C03645=1237.341,-59.055,-37.494,-179.972,5.224,148.895
C03646=1237.346,-59.306,-37.482,-179.974,5.224,148.895
C03647=1237.351,-59.555,-37.469,-179.977,5.224,148.896
C03648=1237.356,-59.805,-37.457,-179.980,5.225,148.897
C03649=1237.361,-60.054,-37.445,-179.982,5.224,148.898
C03650=1237.367,-60.304,-37.433,-179.984,5.224,148.898
C03651=1237.371,-60.553,-37.421,-179.987,5.224,148.899
C03652=1237.376,-60.803,-37.408,-179.989,5.224,148.900
C03653=1237.382,-61.053,-37.396,-179.992,5.224,148.900
C03654=1237.387,-61.302,-37.384,-179.994,5.224,148.901
C03655=1237.392,-61.552,-37.371,-179.996,5.224,148.902
C03656=1237.397,-61.802,-37.359,-179.999,5.223,148.903
C03657=1237.402,-62.052,-37.347,179.999,5.224,148.903
C03658=1237.407,-62.301,-37.334,179.996,5.223,148.904
C03659=1237.412,-62.551,-37.323,179.994,5.223,148.905
C03660=1237.418,-62.801,-37.311,179.991,5.223,148.905
C03661=1237.423,-63.050,-37.299,179.989,5.223,148.906
C03662=1237.428,-63.300,-37.287,179.986,5.223,148.907
C03663=1237.433,-63.549,-37.274,179.984,5.223,148.908
C03664=1237.439,-63.799,-37.262,179.981,5.223,148.908
C03665=1237.443,-64.048,-37.250,179.979,5.223,148.909
C03666=1237.449,-64.298,-37.238,179.977,5.223,148.910
C03667=1237.454,-64.547,-37.226,179.974,5.223,148.911
C03668=1237.459,-64.797,-37.214,179.972,5.223,148.911
C03669=1237.464,-65.047,-37.202,179.970,5.223,148.912
C03670=1237.468,-65.297,-37.190,179.967,5.222,148.913
C03671=1237.474,-65.547,-37.178,179.965,5.223,148.913
C03672=1237.479,-65.796,-37.165,179.962,5.222,148.914
C03673=1237.484,-66.046,-37.153,179.960,5.223,148.915
C03674=1237.490,-66.296,-37.141,179.958,5.222,148.916
C03675=1237.494,-66.545,-37.129,179.955,5.223,148.916
C03676=1237.500,-66.795,-37.117,179.953,5.222,148.917
C03677=1237.505,-67.045,-37.106,179.951,5.222,148.918
C03678=1237.510,-67.294,-37.093,179.948,5.222,148.919
C03679=1237.515,-67.544,-37.082,179.945,5.223,148.919
C03680=1237.520,-67.794,-37.070,179.943,5.222,148.920
C03681=1237.525,-68.043,-37.057,179.941,5.222,148.921
C03682=1237.531,-68.293,-37.045,179.938,5.222,148.921
C03683=1237.535,-68.543,-37.034,179.936,5.222,148.922
C03684=1237.541,-68.792,-37.021,179.933,5.222,148.923
C03685=1237.546,-69.042,-37.010,179.931,5.221,148.924
C03686=1237.551,-69.292,-36.998,179.928,5.222,148.924
C03687=1237.556,-69.541,-36.986,179.926,5.221,148.925
C03688=1237.561,-69.791,-36.974,179.924,5.222,148.926
C03689=1237.567,-70.041,-36.962,179.921,5.221,148.926
C03690=1237.572,-70.291,-36.950,179.919,5.221,148.927
C03691=1237.576,-70.540,-36.938,179.916,5.221,148.928
C03692=1237.582,-70.789,-36.926,179.914,5.221,148.929
C03693=1237.588,-71.039,-36.915,179.912,5.221,148.929
C03694=1237.593,-71.289,-36.903,179.909,5.221,148.930
C03695=1237.598,-71.538,-36.891,179.906,5.221,148.931
C03696=1237.603,-71.788,-36.879,179.904,5.221,148.932
C03697=1237.608,-72.037,-36.867,179.902,5.221,148.932
C03698=1237.613,-72.287,-36.856,179.899,5.221,148.933
C03699=1237.619,-72.537,-36.844,179.897,5.221,148.934
C03700=1237.623,-72.786,-36.832,179.895,5.221,148.934
C03701=1237.629,-73.036,-36.820,179.892,5.221,148.935
C03702=1237.634,-73.286,-36.808,179.890,5.221,148.936
C03703=1237.639,-73.536,-36.797,179.887,5.220,148.937
C03704=1237.644,-73.786,-36.785,179.885,5.221,148.937
C03705=1237.650,-74.055,-36.772,179.882,5.220,148.938
C03706=1237.655,-74.326,-36.759,179.880,5.221,148.939
C03707=1237.661,-74.596,-36.746,179.877,5.221,148.940
C03708=1237.667,-74.866,-36.734,179.875,5.220,148.940
C03709=1237.672,-75.116,-36.722,179.872,5.220,148.941
C03710=1237.677,-75.365,-36.710,179.870,5.220,148.942
C03711=1237.682,-75.615,-36.699,179.868,5.220,148.942
C03712=1237.687,-75.865,-36.687,179.865,5.220,148.943
C03713=1237.692,-76.115,-36.675,179.863,5.220,148.944
C03714=1237.698,-76.365,-36.664,179.860,5.220,148.945
C03715=1237.702,-76.614,-36.652,179.858,5.220,148.945
C03716=1237.708,-76.864,-36.641,179.855,5.220,148.946
C03717=1237.713,-77.113,-36.629,179.853,5.220,148.947
C03718=1237.718,-77.363,-36.618,179.850,5.220,148.948
C03719=1237.723,-77.613,-36.606,179.848,5.220,148.948
C03720=1237.729,-77.863,-36.594,179.845,5.220,148.949
C03721=1237.733,-78.112,-36.583,179.843,5.220,148.950
C03722=1237.739,-78.362,-36.571,179.841,5.220,148.950
C03723=1237.744,-78.612,-36.559,179.839,5.220,148.951
C03724=1237.749,-78.861,-36.548,179.836,5.219,148.952
C03725=1237.755,-79.110,-36.536,179.834,5.220,148.953
C03726=1237.759,-79.360,-36.524,179.831,5.219,148.953
C03727=1237.765,-79.610,-36.513,179.829,5.220,148.954
C03728=1237.769,-79.860,-36.501,179.826,5.219,148.955
C03729=1237.775,-80.110,-36.489,179.824,5.220,148.955
C03730=1237.780,-80.359,-36.479,179.822,5.220,148.956
C03731=1237.786,-80.609,-36.467,179.820,5.219,148.957
C03732=1237.791,-80.859,-36.456,179.817,5.220,148.958
C03733=1237.796,-81.109,-36.444,179.815,5.219,148.958
C03734=1237.801,-81.358,-36.433,179.813,5.220,148.959
C03735=1237.806,-81.608,-36.421,179.810,5.219,148.960
C03736=1237.811,-81.857,-36.410,179.808,5.219,148.960
C03737=1237.816,-82.107,-36.399,179.805,5.219,148.961
C03738=1237.821,-82.357,-36.387,179.803,5.219,148.962
C03739=1237.826,-82.606,-36.376,179.800,5.219,148.963
C03740=1237.832,-82.856,-36.364,179.798,5.220,148.963
C03741=1237.837,-83.105,-36.353,179.795,5.219,148.964
C03742=1237.842,-83.355,-36.341,179.793,5.220,148.965
C03743=1237.847,-83.605,-36.330,179.790,5.219,148.966
C03744=1237.853,-83.855,-36.318,179.788,5.219,148.966
C03745=1237.857,-84.105,-36.307,179.786,5.219,148.967
C03746=1237.863,-84.354,-36.296,179.784,5.219,148.968
C03747=1237.868,-84.604,-36.284,179.781,5.219,148.968
C03748=1237.873,-84.853,-36.273,179.779,5.219,148.969
C03749=1237.878,-85.103,-36.261,179.776,5.219,148.970
C03750=1237.883,-85.353,-36.250,179.774,5.219,148.971
C03751=1237.889,-85.603,-36.240,179.771,5.219,148.971
C03752=1237.894,-85.852,-36.228,179.769,5.219,148.972
C03753=1237.899,-86.102,-36.216,179.767,5.218,148.973
C03754=1237.903,-86.352,-36.205,179.765,5.219,148.973
C03755=1237.909,-86.601,-36.194,179.762,5.218,148.974
C03756=1237.914,-86.851,-36.182,179.760,5.219,148.975
C03757=1237.920,-87.101,-36.171,179.757,5.218,148.976
C03758=1237.925,-87.351,-36.160,179.755,5.219,148.976
C03759=1237.930,-87.600,-36.149,179.752,5.218,148.977
C03760=1237.935,-87.850,-36.137,179.750,5.218,148.978
C03761=1237.940,-88.100,-36.127,179.748,5.219,148.978
C03762=1237.945,-88.349,-36.115,179.745,5.218,148.979
C03763=1237.951,-88.599,-36.104,179.743,5.219,148.980
C03764=1237.956,-88.848,-36.092,179.741,5.218,148.981
C03765=1237.961,-89.099,-36.082,179.739,5.219,148.981
C03766=1237.966,-89.349,-36.070,179.736,5.218,148.982
C03767=1237.971,-89.597,-36.059,179.734,5.218,148.983
C03768=1237.976,-89.847,-36.048,179.731,5.218,148.983
C03769=1237.982,-90.098,-36.037,179.729,5.218,148.984
C03770=1237.987,-90.347,-36.026,179.726,5.218,148.985
C03771=1237.992,-90.596,-36.014,179.724,5.218,148.985
C03772=1237.997,-90.846,-36.004,179.722,5.218,148.986
C03773=1238.003,-91.096,-35.992,179.720,5.218,148.987
C03774=1238.008,-91.345,-35.981,179.716,5.218,148.988
C03775=1238.013,-91.596,-35.970,179.714,5.218,148.989
C03776=1238.018,-91.845,-35.959,179.712,5.218,148.989
C03777=1238.023,-92.094,-35.948,179.710,5.218,148.990
C03778=1238.028,-92.345,-35.937,179.707,5.218,148.991
C03779=1238.033,-92.594,-35.926,179.705,5.218,148.991
C03780=1238.039,-92.843,-35.914,179.702,5.218,148.992
C03781=1238.044,-93.094,-35.904,179.700,5.218,148.993
C03782=1238.049,-93.343,-35.892,179.698,5.218,148.994
C03783=1238.054,-93.593,-35.882,179.695,5.218,148.994
C03784=1238.060,-93.843,-35.870,179.693,5.218,148.995
C03785=1238.064,-94.092,-35.859,179.690,5.218,148.996
C03786=1238.070,-94.342,-35.849,179.688,5.218,148.996
C03787=1238.075,-94.592,-35.837,179.686,5.218,148.997
C03788=1238.080,-94.841,-35.827,179.684,5.218,148.998
C03789=1238.086,-95.091,-35.815,179.681,5.218,148.999
C03790=1238.090,-95.341,-35.804,179.679,5.218,148.999
C03791=1238.096,-95.590,-35.794,179.676,5.218,149.000
C03792=1238.101,-95.840,-35.783,179.674,5.218,149.001
C03793=1238.106,-96.090,-35.772,179.671,5.217,149.001
C03794=1238.112,-96.339,-35.760,179.669,5.218,149.002
C03795=1238.117,-96.590,-35.750,179.667,5.217,149.003
C03796=1238.122,-96.839,-35.739,179.665,5.218,149.004
C03797=1238.127,-97.089,-35.728,179.662,5.218,149.004
C03798=1238.132,-97.338,-35.717,179.660,5.218,149.005
C03799=1238.137,-97.588,-35.707,179.658,5.218,149.006
C03800=1238.143,-97.838,-35.695,179.655,5.217,149.006
C03801=1238.148,-98.088,-35.684,179.653,5.218,149.007
C03802=1238.153,-98.337,-35.674,179.650,5.217,149.008
C03803=1238.158,-98.587,-35.663,179.648,5.218,149.009
C03804=1238.163,-98.836,-35.652,179.645,5.217,149.009
C03805=1238.168,-99.087,-35.641,179.643,5.218,149.010
C03806=1238.174,-99.335,-35.631,179.641,5.217,149.011
C03807=1238.179,-99.586,-35.619,179.639,5.218,149.011
C03808=1238.184,-99.836,-35.608,179.636,5.217,149.012
C03809=1238.190,-100.106,-35.598,179.634,5.217,149.013
C03810=1238.195,-100.377,-35.585,179.631,5.217,149.014
C03811=1238.200,-100.648,-35.574,179.629,5.218,149.014
C03812=1238.207,-100.919,-35.562,179.626,5.217,149.015
C03813=1238.212,-101.168,-35.551,179.624,5.218,149.016
C03814=1238.217,-101.419,-35.541,179.621,5.217,149.017
C03815=1238.222,-101.668,-35.530,179.619,5.218,149.017
C03816=1238.227,-101.918,-35.519,179.616,5.217,149.018
C03817=1238.232,-102.167,-35.509,179.614,5.217,149.019
C03818=1238.238,-102.417,-35.497,179.612,5.217,149.019
C03819=1238.243,-102.667,-35.487,179.609,5.217,149.020
C03820=1238.248,-102.917,-35.476,179.607,5.217,149.021
C03821=1238.254,-103.166,-35.465,179.605,5.217,149.022
C03822=1238.259,-103.416,-35.455,179.602,5.217,149.022
C03823=1238.264,-103.666,-35.444,179.600,5.217,149.023
C03824=1238.269,-103.915,-35.433,179.598,5.218,149.024
C03825=1238.275,-104.165,-35.423,179.595,5.217,149.024
C03826=1238.280,-104.415,-35.412,179.593,5.217,149.025
C03827=1238.284,-104.665,-35.401,179.590,5.217,149.026
C03828=1238.290,-104.914,-35.391,179.588,5.217,149.027
C03829=1238.295,-105.165,-35.380,179.586,5.217,149.027
C03830=1238.300,-105.414,-35.369,179.584,5.217,149.028
C03831=1238.305,-105.664,-35.359,179.581,5.217,149.029
C03832=1238.311,-105.913,-35.349,179.579,5.217,149.029
C03833=1238.316,-106.164,-35.338,179.576,5.217,149.030
C03834=1238.321,-106.412,-35.327,179.574,5.217,149.031
C03835=1238.326,-106.663,-35.317,179.572,5.217,149.031
C03836=1238.332,-106.912,-35.306,179.570,5.217,149.032
C03837=1238.337,-107.163,-35.296,179.568,5.217,149.033
C03838=1238.342,-107.411,-35.285,179.565,5.217,149.034
C03839=1238.348,-107.661,-35.275,179.563,5.217,149.034
C03840=1238.353,-107.911,-35.264,179.560,5.216,149.035
C03841=1238.358,-108.161,-35.254,179.558,5.217,149.036
C03842=1238.362,-108.410,-35.243,179.555,5.216,149.036
C03843=1238.368,-108.660,-35.233,179.553,5.217,149.037
C03844=1238.373,-108.910,-35.222,179.551,5.216,149.038
C03845=1238.378,-109.159,-35.212,179.549,5.217,149.039
C03846=1238.383,-109.410,-35.202,179.546,5.217,149.039
C03847=1238.389,-109.659,-35.191,179.544,5.217,149.040
C03848=1238.394,-109.909,-35.180,179.542,5.217,149.041
C03849=1238.399,-110.158,-35.170,179.539,5.217,149.041
C03850=1238.404,-110.409,-35.159,179.537,5.217,149.042
C03851=1238.410,-110.658,-35.149,179.534,5.216,149.043
C03852=1238.415,-110.908,-35.139,179.532,5.217,149.044
C03853=1238.420,-111.158,-35.128,179.529,5.216,149.044
C03854=1238.425,-111.407,-35.119,179.527,5.217,149.045
C03855=1238.430,-111.657,-35.107,179.525,5.217,149.046
C03856=1238.436,-111.906,-35.097,179.523,5.217,149.046
C03857=1238.441,-112.157,-35.087,179.520,5.217,149.047
C03858=1238.446,-112.406,-35.076,179.518,5.217,149.048
C03859=1238.452,-112.656,-35.066,179.516,5.217,149.049
C03860=1238.457,-112.906,-35.056,179.513,5.216,149.049
C03861=1238.462,-113.155,-35.045,179.511,5.217,149.050
C03862=1238.467,-113.405,-35.035,179.508,5.216,149.051
C03863=1238.472,-113.655,-35.025,179.506,5.217,149.051
C03864=1238.478,-113.904,-35.015,179.503,5.216,149.052
C03865=1238.483,-114.155,-35.004,179.501,5.217,149.053
C03866=1238.488,-114.404,-34.994,179.500,5.217,149.053
C03867=1238.494,-114.653,-34.983,179.497,5.216,149.054
C03868=1238.498,-114.903,-34.973,179.495,5.217,149.055
C03869=1238.504,-115.153,-34.963,179.492,5.216,149.055
C03870=1238.509,-115.403,-34.953,179.490,5.217,149.056
C03871=1238.514,-115.652,-34.942,179.488,5.216,149.057
C03872=1238.520,-115.902,-34.932,179.485,5.216,149.058
C03873=1238.524,-116.152,-34.922,179.483,5.216,149.058
C03874=1238.530,-116.401,-34.912,179.481,5.216,149.059
C03875=1238.535,-116.651,-34.902,179.479,5.217,149.060
C03876=1238.540,-116.901,-34.891,179.476,5.216,149.060
C03877=1238.546,-117.151,-34.881,179.474,5.217,149.061
C03878=1238.550,-117.401,-34.871,179.471,5.216,149.062
C03879=1238.556,-117.651,-34.861,179.469,5.217,149.063
C03880=1238.562,-117.900,-34.851,179.466,5.216,149.063
C03881=1238.567,-118.151,-34.841,179.464,5.217,149.064
C03882=1238.571,-118.400,-34.831,179.462,5.216,149.065
C03883=1238.577,-118.649,-34.821,179.459,5.216,149.065
C03884=1238.582,-118.900,-34.810,179.457,5.217,149.066
C03885=1238.588,-119.149,-34.800,179.455,5.216,149.067
C03886=1238.592,-119.398,-34.790,179.453,5.216,149.067
C03887=1238.597,-119.649,-34.780,179.450,5.216,149.068
C03888=1238.603,-119.898,-34.770,179.448,5.216,149.069
C03889=1238.608,-120.148,-34.760,179.446,5.216,149.070
C03890=1238.613,-120.397,-34.750,179.444,5.216,149.070
C03891=1238.619,-120.648,-34.740,179.441,5.216,149.071
C03892=1238.624,-120.897,-34.730,179.439,5.216,149.072
C03893=1238.629,-121.147,-34.720,179.437,5.217,149.072
C03894=1238.634,-121.397,-34.710,179.434,5.216,149.073
C03895=1238.640,-121.646,-34.699,179.432,5.216,149.074
C03896=1238.645,-121.896,-34.690,179.429,5.216,149.075
C03897=1238.650,-122.146,-34.679,179.427,5.216,149.075
C03898=1238.656,-122.396,-34.670,179.424,5.216,149.076
C03899=1238.660,-122.645,-34.660,179.422,5.216,149.077
C03900=1238.666,-122.895,-34.650,179.421,5.216,149.077
C03901=1238.671,-123.145,-34.639,179.418,5.216,149.078
C03902=1238.676,-123.394,-34.630,179.416,5.216,149.079
C03903=1238.682,-123.644,-34.620,179.413,5.216,149.079
C03904=1238.687,-123.895,-34.610,179.411,5.216,149.080
C03905=1238.692,-124.144,-34.600,179.408,5.216,149.081
C03906=1238.697,-124.394,-34.590,179.406,5.216,149.082
C03907=1238.702,-124.643,-34.580,179.404,5.216,149.082
C03908=1238.707,-124.894,-34.570,179.402,5.216,149.083
C03909=1238.713,-125.143,-34.560,179.400,5.216,149.084
C03910=1238.718,-125.392,-34.551,179.397,5.216,149.084
C03911=1238.724,-125.642,-34.540,179.395,5.216,149.085
C03912=1238.729,-125.893,-34.530,179.393,5.216,149.086
C03913=1238.307,-125.903,-34.566,179.388,5.219,149.088
C03914=1238.302,-125.653,-34.575,179.391,5.220,149.087
C03915=1238.297,-125.403,-34.586,179.393,5.219,149.086
C03916=1238.292,-125.154,-34.595,179.395,5.219,149.086
C03917=1238.286,-124.904,-34.605,179.397,5.220,149.085
C03918=1238.280,-124.654,-34.615,179.399,5.219,149.084
C03919=1238.276,-124.404,-34.625,179.402,5.220,149.084
C03920=1238.270,-124.154,-34.635,179.404,5.219,149.083
C03921=1238.265,-123.905,-34.645,179.407,5.220,149.082
C03922=1238.260,-123.655,-34.654,179.409,5.219,149.081
C03923=1238.255,-123.405,-34.665,179.411,5.220,149.081
C03924=1238.250,-123.156,-34.674,179.414,5.219,149.080
C03925=1238.244,-122.906,-34.685,179.416,5.219,149.079
C03926=1238.239,-122.656,-34.695,179.418,5.219,149.079
C03927=1238.234,-122.406,-34.704,179.420,5.219,149.078
C03928=1238.228,-122.156,-34.714,179.423,5.220,149.077
C03929=1238.223,-121.907,-34.724,179.425,5.220,149.077
C03930=1238.219,-121.657,-34.734,179.427,5.220,149.076
C03931=1238.213,-121.407,-34.745,179.429,5.220,149.075
C03932=1238.207,-121.158,-34.755,179.432,5.220,149.075
C03933=1238.201,-120.908,-34.764,179.434,5.220,149.074
C03934=1238.197,-120.658,-34.774,179.436,5.219,149.073
C03935=1238.192,-120.408,-34.785,179.439,5.220,149.072
C03936=1238.186,-120.159,-34.795,179.441,5.219,149.072
C03937=1238.182,-119.909,-34.805,179.444,5.220,149.071
C03938=1238.176,-119.659,-34.815,179.446,5.219,149.070
C03939=1238.171,-119.410,-34.825,179.449,5.220,149.070
C03940=1238.166,-119.159,-34.836,179.451,5.220,149.069
C03941=1238.161,-118.910,-34.845,179.453,5.219,149.068
C03942=1238.155,-118.660,-34.855,179.455,5.220,149.067
C03943=1238.150,-118.410,-34.865,179.458,5.219,149.067
C03944=1238.145,-118.161,-34.875,179.460,5.220,149.066
C03945=1238.139,-117.911,-34.885,179.462,5.220,149.065
C03946=1238.134,-117.661,-34.896,179.465,5.220,149.065
C03947=1238.129,-117.411,-34.906,179.467,5.220,149.064
C03948=1238.124,-117.162,-34.916,179.469,5.220,149.063
C03949=1238.119,-116.912,-34.926,179.471,5.220,149.063
C03950=1238.113,-116.662,-34.936,179.473,5.219,149.062
C03951=1238.108,-116.413,-34.947,179.476,5.220,149.061
C03952=1238.103,-116.162,-34.957,179.478,5.220,149.060
C03953=1238.098,-115.913,-34.967,179.481,5.220,149.060
C03954=1238.092,-115.664,-34.977,179.483,5.220,149.059
C03955=1238.087,-115.413,-34.988,179.486,5.220,149.058
C03956=1238.082,-115.164,-34.998,179.488,5.220,149.058
C03957=1238.077,-114.914,-35.008,179.491,5.220,149.057
C03958=1238.072,-114.664,-35.018,179.493,5.220,149.056
C03959=1238.066,-114.415,-35.028,179.495,5.220,149.055
C03960=1238.061,-114.165,-35.039,179.497,5.220,149.055
C03961=1238.056,-113.915,-35.049,179.499,5.219,149.054
C03962=1238.050,-113.665,-35.059,179.502,5.220,149.053
C03963=1238.045,-113.415,-35.070,179.504,5.220,149.053
C03964=1238.040,-113.166,-35.079,179.506,5.220,149.052
C03965=1238.035,-112.916,-35.090,179.509,5.220,149.051
C03966=1238.030,-112.667,-35.101,179.511,5.220,149.051
C03967=1238.024,-112.417,-35.111,179.513,5.220,149.050
C03968=1238.019,-112.167,-35.122,179.516,5.220,149.049
C03969=1238.014,-111.917,-35.132,179.518,5.220,149.049
C03970=1238.009,-111.667,-35.142,179.520,5.220,149.048
C03971=1238.004,-111.418,-35.152,179.523,5.220,149.047
C03972=1237.999,-111.168,-35.163,179.525,5.220,149.046
C03973=1237.993,-110.918,-35.173,179.528,5.220,149.046
C03974=1237.988,-110.669,-35.183,179.530,5.220,149.045
C03975=1237.983,-110.419,-35.194,179.532,5.220,149.044
C03976=1237.977,-110.170,-35.205,179.534,5.220,149.044
C03977=1237.972,-109.919,-35.215,179.537,5.220,149.043
C03978=1237.967,-109.670,-35.225,179.539,5.220,149.042
C03979=1237.962,-109.419,-35.236,179.541,5.220,149.041
C03980=1237.956,-109.170,-35.246,179.544,5.220,149.041
C03981=1237.952,-108.921,-35.256,179.546,5.220,149.040
C03982=1237.947,-108.671,-35.267,179.549,5.220,149.039
C03983=1237.941,-108.422,-35.277,179.551,5.220,149.038
C03984=1237.936,-108.171,-35.288,179.554,5.220,149.038
C03985=1237.930,-107.922,-35.298,179.556,5.220,149.037
C03986=1237.926,-107.672,-35.309,179.558,5.220,149.036
C03987=1237.920,-107.423,-35.320,179.560,5.220,149.036
C03988=1237.915,-107.172,-35.330,179.563,5.220,149.035
C03989=1237.909,-106.923,-35.340,179.565,5.220,149.034
C03990=1237.904,-106.673,-35.351,179.567,5.220,149.033
C03991=1237.899,-106.424,-35.362,179.570,5.220,149.033
C03992=1237.894,-106.173,-35.372,179.572,5.220,149.032
C03993=1237.889,-105.924,-35.383,179.574,5.221,149.032
C03994=1237.884,-105.674,-35.394,179.576,5.220,149.031
C03995=1237.878,-105.425,-35.404,179.579,5.221,149.030
C03996=1237.873,-105.174,-35.415,179.581,5.220,149.029
C03997=1237.868,-104.925,-35.425,179.584,5.221,149.029
C03998=1237.863,-104.675,-35.436,179.586,5.221,149.028
C03999=1237.857,-104.426,-35.446,179.589,5.221,149.027
C04000=1237.852,-104.175,-35.457,179.591,5.221,149.027
C04001=1237.847,-103.927,-35.468,179.593,5.221,149.026
C04002=1237.842,-103.676,-35.478,179.595,5.221,149.025
C04003=1237.836,-103.427,-35.489,179.598,5.220,149.024
C04004=1237.832,-103.177,-35.500,179.600,5.221,149.024
C04005=1237.826,-102.928,-35.510,179.602,5.220,149.023
C04006=1237.821,-102.677,-35.521,179.605,5.221,149.022
C04007=1237.816,-102.428,-35.532,179.607,5.221,149.022
C04008=1237.811,-102.178,-35.542,179.610,5.221,149.021
C04009=1237.806,-101.928,-35.553,179.612,5.221,149.020
C04010=1237.801,-101.679,-35.564,179.615,5.221,149.019
C04011=1237.796,-101.429,-35.574,179.617,5.221,149.019
C04012=1237.790,-101.180,-35.585,179.619,5.221,149.018
C04013=1237.785,-100.929,-35.596,179.621,5.221,149.017
C04014=1237.779,-100.659,-35.608,179.624,5.221,149.017
C04015=1237.773,-100.388,-35.619,179.627,5.220,149.016
C04016=1237.768,-100.117,-35.631,179.629,5.221,149.015
C04017=1237.763,-99.846,-35.643,179.631,5.221,149.014
C04018=1237.757,-99.597,-35.653,179.634,5.221,149.013
C04019=1237.752,-99.347,-35.665,179.636,5.221,149.013
C04020=1237.747,-99.097,-35.675,179.639,5.221,149.012
C04021=1237.742,-98.847,-35.685,179.641,5.221,149.011
C04022=1237.736,-98.598,-35.697,179.644,5.221,149.011
C04023=1237.731,-98.348,-35.708,179.646,5.221,149.010
C04024=1237.726,-98.098,-35.719,179.648,5.221,149.009
C04025=1237.720,-97.848,-35.729,179.651,5.221,149.009
C04026=1237.716,-97.599,-35.740,179.653,5.221,149.008
C04027=1237.710,-97.349,-35.751,179.655,5.221,149.007
C04028=1237.706,-97.100,-35.762,179.657,5.221,149.006
C04029=1237.700,-96.849,-35.773,179.660,5.221,149.006
C04030=1237.694,-96.600,-35.784,179.662,5.221,149.005
C04031=1237.689,-96.350,-35.794,179.665,5.221,149.004
C04032=1237.685,-96.100,-35.806,179.667,5.221,149.004
C04033=1237.679,-95.851,-35.816,179.670,5.221,149.003
C04034=1237.674,-95.601,-35.828,179.672,5.221,149.002
C04035=1237.668,-95.352,-35.839,179.674,5.221,149.001
C04036=1237.663,-95.102,-35.849,179.676,5.221,149.001
C04037=1237.659,-94.852,-35.861,179.679,5.222,149.000
C04038=1237.653,-94.602,-35.871,179.681,5.221,148.999
C04039=1237.648,-94.353,-35.883,179.684,5.222,148.999
C04040=1237.643,-94.102,-35.893,179.686,5.221,148.998
C04041=1237.637,-93.853,-35.904,179.689,5.222,148.997
C04042=1237.633,-93.604,-35.916,179.691,5.221,148.996
C04043=1237.628,-93.353,-35.926,179.693,5.222,148.996
C04044=1237.622,-93.104,-35.938,179.696,5.222,148.995
C04045=1237.617,-92.854,-35.948,179.698,5.221,148.994
C04046=1237.612,-92.604,-35.959,179.700,5.222,148.994
C04047=1237.607,-92.355,-35.970,179.702,5.221,148.993
C04048=1237.601,-92.105,-35.982,179.705,5.222,148.992
C04049=1237.596,-91.855,-35.993,179.707,5.221,148.991
C04050=1237.591,-91.606,-36.004,179.710,5.222,148.991
C04051=1237.585,-91.356,-36.015,179.712,5.222,148.990
C04052=1237.581,-91.106,-36.026,179.715,5.222,148.989
C04053=1237.575,-90.857,-36.037,179.717,5.222,148.989
C04054=1237.570,-90.607,-36.048,179.719,5.222,148.988
C04055=1237.565,-90.357,-36.060,179.721,5.222,148.987
C04056=1237.560,-90.108,-36.071,179.724,5.222,148.986
C04057=1237.555,-89.858,-36.081,179.726,5.222,148.986
C04058=1237.549,-89.608,-36.093,179.729,5.222,148.985
C04059=1237.544,-89.358,-36.104,179.731,5.222,148.984
C04060=1237.539,-89.109,-36.115,179.734,5.222,148.984
C04061=1237.534,-88.859,-36.126,179.736,5.222,148.983
C04062=1237.529,-88.609,-36.138,179.739,5.222,148.982
C04063=1237.523,-88.360,-36.149,179.741,5.222,148.981
C04064=1237.518,-88.110,-36.159,179.743,5.221,148.981
C04065=1237.513,-87.860,-36.171,179.746,5.222,148.980
C04066=1237.508,-87.611,-36.182,179.748,5.222,148.979
C04067=1237.502,-87.361,-36.194,179.751,5.222,148.978
C04068=1237.498,-87.112,-36.205,179.753,5.222,148.978
C04069=1237.493,-86.861,-36.216,179.755,5.222,148.977
C04070=1237.487,-86.611,-36.228,179.757,5.222,148.976
C04071=1237.482,-86.363,-36.239,179.760,5.222,148.976
C04072=1237.477,-86.113,-36.250,179.762,5.222,148.975
C04073=1237.472,-85.863,-36.262,179.765,5.222,148.974
C04074=1237.467,-85.613,-36.272,179.767,5.222,148.973
C04075=1237.461,-85.364,-36.283,179.770,5.222,148.973
C04076=1237.456,-85.114,-36.295,179.772,5.222,148.972
C04077=1237.451,-84.864,-36.306,179.774,5.223,148.971
C04078=1237.446,-84.614,-36.318,179.776,5.222,148.971
C04079=1237.441,-84.365,-36.330,179.779,5.223,148.970
C04080=1237.436,-84.115,-36.340,179.781,5.222,148.969
C04081=1237.430,-83.865,-36.352,179.784,5.223,148.968
C04082=1237.426,-83.616,-36.363,179.786,5.222,148.968
C04083=1237.420,-83.366,-36.375,179.789,5.223,148.967
C04084=1237.415,-83.117,-36.386,179.791,5.223,148.966
C04085=1237.409,-82.867,-36.398,179.793,5.223,148.966
C04086=1237.405,-82.617,-36.409,179.796,5.223,148.965
C04087=1237.400,-82.368,-36.420,179.798,5.223,148.964
C04088=1237.395,-82.118,-36.432,179.800,5.223,148.963
C04089=1237.390,-81.867,-36.443,179.803,5.223,148.963
C04090=1237.384,-81.618,-36.454,179.805,5.223,148.962
C04091=1237.379,-81.368,-36.466,179.808,5.223,148.961
C04092=1237.373,-81.119,-36.477,179.810,5.223,148.961
C04093=1237.369,-80.869,-36.489,179.812,5.224,148.960
C04094=1237.363,-80.619,-36.501,179.815,5.223,148.959
C04095=1237.358,-80.370,-36.511,179.818,5.223,148.958
C04096=1237.353,-80.120,-36.523,179.820,5.223,148.958
C04097=1237.348,-79.871,-36.535,179.823,5.223,148.957
C04098=1237.342,-79.621,-36.547,179.825,5.223,148.956
C04099=1237.338,-79.371,-36.558,179.827,5.223,148.955
C04100=1237.332,-79.121,-36.570,179.829,5.223,148.955
C04101=1237.328,-78.871,-36.581,179.831,5.223,148.954
C04102=1237.322,-78.622,-36.593,179.834,5.223,148.953
C04103=1237.317,-78.373,-36.604,179.836,5.223,148.953
C04104=1237.311,-78.123,-36.616,179.839,5.223,148.952
C04105=1237.307,-77.873,-36.627,179.841,5.223,148.951
C04106=1237.301,-77.623,-36.639,179.844,5.224,148.950
C04107=1237.297,-77.373,-36.650,179.846,5.223,148.950
C04108=1237.291,-77.123,-36.662,179.848,5.224,148.949
C04109=1237.285,-76.874,-36.674,179.851,5.223,148.948
C04110=1237.281,-76.625,-36.685,179.853,5.224,148.948
C04111=1237.275,-76.375,-36.697,179.855,5.224,148.947
C04112=1237.271,-76.126,-36.709,179.858,5.224,148.946
C04113=1237.265,-75.876,-36.721,179.860,5.224,148.945
C04114=1237.261,-75.626,-36.732,179.863,5.224,148.945
C04115=1237.255,-75.376,-36.744,179.865,5.224,148.944
C04116=1237.250,-75.126,-36.756,179.867,5.224,148.943
C04117=1237.245,-74.877,-36.767,179.870,5.224,148.943
C04118=1237.239,-74.607,-36.780,179.873,5.224,148.942
C04119=1237.234,-74.337,-36.793,179.875,5.224,148.941
C04120=1237.228,-74.066,-36.804,179.877,5.224,148.940
C04121=1237.222,-73.796,-36.817,179.881,5.224,148.939
C04122=1237.217,-73.546,-36.829,179.883,5.224,148.939
C04123=1237.212,-73.297,-36.842,179.885,5.224,148.938
C04124=1237.207,-73.047,-36.853,179.888,5.224,148.937
C04125=1237.202,-72.797,-36.865,179.890,5.225,148.937
C04126=1237.197,-72.548,-36.876,179.892,5.224,148.936
C04127=1237.191,-72.298,-36.888,179.895,5.225,148.935
C04128=1237.186,-72.048,-36.900,179.897,5.224,148.934
C04129=1237.182,-71.799,-36.912,179.900,5.225,148.934
C04130=1237.176,-71.549,-36.924,179.902,5.224,148.933
C04131=1237.170,-71.299,-36.936,179.904,5.225,148.932
C04132=1237.165,-71.050,-36.947,179.907,5.225,148.932
C04133=1237.160,-70.801,-36.959,179.909,5.225,148.931
C04134=1237.155,-70.551,-36.971,179.911,5.225,148.930
C04135=1237.150,-70.301,-36.983,179.914,5.225,148.929
C04136=1237.145,-70.051,-36.994,179.917,5.226,148.929
C04137=1237.140,-69.802,-37.007,179.919,5.225,148.928
C04138=1237.134,-69.552,-37.019,179.922,5.225,148.927
C04139=1237.130,-69.302,-37.030,179.924,5.225,148.926
C04140=1237.124,-69.052,-37.042,179.927,5.226,148.926
C04141=1237.119,-68.803,-37.055,179.929,5.225,148.925
C04142=1237.114,-68.553,-37.067,179.931,5.226,148.924
C04143=1237.109,-68.303,-37.078,179.934,5.225,148.924
C04144=1237.104,-68.054,-37.091,179.936,5.226,148.923
C04145=1237.098,-67.804,-37.102,179.938,5.226,148.922
C04146=1237.093,-67.554,-37.114,179.941,5.226,148.921
C04147=1237.088,-67.305,-37.126,179.943,5.226,148.921
C04148=1237.083,-67.055,-37.138,179.946,5.226,148.920
C04149=1237.078,-66.805,-37.150,179.948,5.226,148.919
C04150=1237.073,-66.556,-37.163,179.950,5.226,148.919
C04151=1237.068,-66.306,-37.174,179.953,5.226,148.918
C04152=1237.062,-66.056,-37.186,179.955,5.226,148.917
C04153=1237.057,-65.807,-37.198,179.957,5.226,148.916
C04154=1237.052,-65.557,-37.210,179.960,5.227,148.916
C04155=1237.046,-65.307,-37.222,179.963,5.226,148.915
C04156=1237.042,-65.058,-37.234,179.965,5.226,148.914
C04157=1237.037,-64.808,-37.246,179.967,5.226,148.913
C04158=1237.032,-64.559,-37.259,179.970,5.227,148.913
C04159=1237.026,-64.309,-37.271,179.972,5.226,148.912
C04160=1237.021,-64.059,-37.282,179.975,5.227,148.911
C04161=1237.016,-63.810,-37.294,179.977,5.226,148.911
C04162=1237.011,-63.559,-37.307,179.980,5.227,148.910
C04163=1237.006,-63.310,-37.319,179.982,5.227,148.909
C04164=1237.001,-63.060,-37.331,179.984,5.227,148.908
C04165=1236.996,-62.811,-37.344,179.986,5.227,148.908
C04166=1236.990,-62.561,-37.356,179.989,5.227,148.907
C04167=1236.986,-62.312,-37.368,179.992,5.228,148.906
C04168=1236.981,-62.062,-37.380,179.994,5.227,148.906
C04169=1236.975,-61.813,-37.392,179.996,5.228,148.905
C04170=1236.970,-61.563,-37.404,179.999,5.227,148.904
C04171=1236.965,-61.313,-37.416,-179.998,5.228,148.903
C04172=1236.959,-61.063,-37.429,-179.996,5.227,148.903
C04173=1236.954,-60.814,-37.441,-179.994,5.228,148.902
C04174=1236.949,-60.563,-37.453,-179.991,5.227,148.901
C04175=1236.945,-60.314,-37.465,-179.989,5.228,148.900
C04176=1236.940,-60.065,-37.477,-179.987,5.228,148.900
C04177=1236.935,-59.815,-37.490,-179.984,5.228,148.899
C04178=1236.929,-59.565,-37.502,-179.982,5.228,148.898
C04179=1236.924,-59.316,-37.514,-179.979,5.228,148.898
C04180=1236.919,-59.066,-37.526,-179.977,5.228,148.897
C04181=1236.913,-58.817,-37.539,-179.975,5.228,148.896
C04182=1236.908,-58.567,-37.551,-179.972,5.228,148.896
C04183=1236.903,-58.317,-37.564,-179.970,5.228,148.895
C04184=1236.898,-58.067,-37.576,-179.967,5.229,148.894
C04185=1236.893,-57.818,-37.588,-179.965,5.229,148.893
C04186=1236.888,-57.568,-37.601,-179.962,5.229,148.893
C04187=1236.883,-57.319,-37.612,-179.960,5.228,148.892
C04188=1236.878,-57.069,-37.625,-179.957,5.229,148.891
C04189=1236.873,-56.820,-37.637,-179.955,5.229,148.890
C04190=1236.868,-56.569,-37.650,-179.952,5.229,148.890
C04191=1236.863,-56.320,-37.662,-179.950,5.229,148.889
C04192=1236.858,-56.071,-37.675,-179.948,5.229,148.888
C04193=1236.852,-55.821,-37.687,-179.945,5.229,148.888
C04194=1236.847,-55.571,-37.699,-179.943,5.229,148.887
C04195=1236.842,-55.322,-37.712,-179.941,5.229,148.886
C04196=1236.837,-55.071,-37.724,-179.938,5.230,148.885
C04197=1236.832,-54.822,-37.737,-179.936,5.229,148.885
C04198=1236.827,-54.573,-37.749,-179.933,5.230,148.884
C04199=1236.822,-54.323,-37.761,-179.931,5.230,148.883
C04200=1236.816,-54.074,-37.774,-179.929,5.230,148.883
C04201=1236.812,-53.824,-37.787,-179.925,5.230,148.882
C04202=1236.807,-53.574,-37.799,-179.923,5.230,148.881
C04203=1236.801,-53.324,-37.811,-179.921,5.230,148.880
C04204=1236.796,-53.075,-37.824,-179.919,5.230,148.880
C04205=1236.791,-52.826,-37.836,-179.916,5.230,148.879
C04206=1236.787,-52.576,-37.849,-179.914,5.230,148.878
C04207=1236.781,-52.326,-37.861,-179.911,5.231,148.877
C04208=1236.775,-52.076,-37.875,-179.909,5.230,148.877
C04209=1236.770,-51.827,-37.887,-179.906,5.231,148.876
C04210=1236.765,-51.577,-37.900,-179.904,5.231,148.875
C04211=1236.760,-51.327,-37.912,-179.902,5.231,148.875
C04212=1236.755,-51.077,-37.925,-179.899,5.231,148.874
C04213=1236.750,-50.828,-37.937,-179.897,5.231,148.873
C04214=1236.745,-50.579,-37.950,-179.894,5.232,148.873
C04215=1236.740,-50.329,-37.963,-179.892,5.231,148.872
C04216=1236.735,-50.079,-37.975,-179.889,5.231,148.871
C04217=1236.730,-49.830,-37.987,-179.887,5.231,148.870
C04218=1236.725,-49.580,-38.000,-179.884,5.231,148.870
C04219=1236.719,-49.330,-38.013,-179.882,5.231,148.869
C04220=1236.714,-49.081,-38.026,-179.879,5.232,148.868
C04221=1236.709,-48.831,-38.039,-179.877,5.232,148.867
C04222=1236.704,-48.561,-38.052,-179.875,5.232,148.867
C04223=1236.698,-48.292,-38.065,-179.872,5.232,148.866
C04224=1236.693,-48.022,-38.079,-179.869,5.232,148.865
C04225=1236.688,-47.752,-38.093,-179.867,5.232,148.864
C04226=1236.682,-47.503,-38.106,-179.864,5.233,148.864
C04227=1236.677,-47.253,-38.119,-179.862,5.232,148.863
C04228=1236.672,-47.003,-38.132,-179.859,5.233,148.862
C04229=1236.667,-46.754,-38.144,-179.856,5.233,148.861
C04230=1236.662,-46.505,-38.157,-179.854,5.233,148.861
C04231=1236.657,-46.255,-38.169,-179.851,5.233,148.860
C04232=1236.651,-46.005,-38.183,-179.849,5.233,148.859
C04233=1236.646,-45.756,-38.196,-179.847,5.233,148.859
C04234=1236.641,-45.506,-38.207,-179.845,5.233,148.858
C04235=1236.636,-45.256,-38.220,-179.842,5.233,148.857
C04236=1236.631,-45.006,-38.233,-179.840,5.233,148.856
C04237=1236.625,-44.757,-38.246,-179.837,5.234,148.856
C04238=1236.621,-44.507,-38.259,-179.835,5.234,148.855
C04239=1236.616,-44.257,-38.272,-179.832,5.234,148.854
C04240=1236.611,-44.008,-38.284,-179.830,5.234,148.854
C04241=1236.605,-43.758,-38.298,-179.828,5.234,148.853
C04242=1236.600,-43.508,-38.311,-179.825,5.235,148.852
C04243=1236.595,-43.259,-38.323,-179.822,5.234,148.851
C04244=1236.590,-43.010,-38.336,-179.820,5.234,148.851
C04245=1236.585,-42.759,-38.349,-179.817,5.235,148.850
C04246=1236.580,-42.510,-38.362,-179.815,5.235,148.849
C04247=1236.575,-42.261,-38.376,-179.812,5.235,148.848
C04248=1236.570,-42.011,-38.388,-179.810,5.235,148.848
C04249=1236.564,-41.762,-38.401,-179.808,5.235,148.847
C04250=1236.560,-41.512,-38.414,-179.806,5.235,148.846
C04251=1236.555,-41.262,-38.427,-179.803,5.235,148.846
C04252=1236.550,-41.013,-38.440,-179.800,5.236,148.845
C04253=1236.544,-40.763,-38.453,-179.798,5.236,148.844
C04254=1236.539,-40.513,-38.466,-179.795,5.236,148.844
C04255=1236.534,-40.264,-38.478,-179.793,5.236,148.843
C04256=1236.529,-40.014,-38.492,-179.791,5.236,148.842
C04257=1236.524,-39.764,-38.504,-179.788,5.236,148.841
C04258=1236.519,-39.515,-38.518,-179.785,5.236,148.841
C04259=1236.514,-39.265,-38.531,-179.783,5.237,148.840
C04260=1236.508,-39.016,-38.544,-179.781,5.236,148.839
C04261=1236.504,-38.766,-38.557,-179.778,5.237,148.838
C04262=1236.498,-38.516,-38.570,-179.776,5.236,148.838
C04263=1236.494,-38.266,-38.583,-179.773,5.237,148.837
C04264=1236.488,-38.017,-38.596,-179.771,5.237,148.836
C04265=1236.483,-37.768,-38.610,-179.769,5.237,148.836
C04266=1236.478,-37.518,-38.623,-179.766,5.238,148.835
C04267=1236.473,-37.269,-38.635,-179.764,5.237,148.834
C04268=1236.468,-37.018,-38.649,-179.761,5.238,148.834
C04269=1236.463,-36.769,-38.661,-179.759,5.238,148.833
C04270=1236.457,-36.520,-38.675,-179.756,5.238,148.832
C04271=1236.453,-36.270,-38.688,-179.753,5.238,148.831
C04272=1236.448,-36.021,-38.701,-179.751,5.238,148.830
C04273=1236.442,-35.770,-38.714,-179.748,5.238,148.830
C04274=1236.437,-35.521,-38.727,-179.746,5.238,148.829
C04275=1236.432,-35.271,-38.741,-179.744,5.239,148.828
C04276=1236.427,-35.022,-38.754,-179.742,5.238,148.828
C04277=1236.422,-34.773,-38.766,-179.739,5.239,148.827
C04278=1236.417,-34.523,-38.781,-179.736,5.239,148.826
C04279=1236.412,-34.274,-38.793,-179.734,5.239,148.826
C04280=1236.407,-34.023,-38.807,-179.732,5.239,148.825
C04281=1236.402,-33.774,-38.819,-179.730,5.239,148.824
C04282=1236.397,-33.524,-38.834,-179.727,5.240,148.823
C04283=1236.392,-33.275,-38.846,-179.724,5.240,148.823
C04284=1236.386,-33.025,-38.860,-179.722,5.239,148.822
C04285=1236.381,-32.776,-38.873,-179.719,5.240,148.821
C04286=1236.376,-32.526,-38.887,-179.717,5.240,148.820
C04287=1236.371,-32.276,-38.899,-179.714,5.240,148.820
C04288=1236.367,-32.027,-38.913,-179.712,5.241,148.819
C04289=1236.361,-31.777,-38.926,-179.709,5.240,148.818
C04290=1236.356,-31.527,-38.939,-179.707,5.241,148.818
C04291=1236.351,-31.278,-38.953,-179.705,5.241,148.817
C04292=1236.346,-31.028,-38.966,-179.702,5.241,148.816
C04293=1236.341,-30.779,-38.979,-179.699,5.242,148.816
C04294=1236.336,-30.529,-38.993,-179.697,5.241,148.815
C04295=1236.330,-30.280,-39.006,-179.695,5.242,148.814
C04296=1236.326,-30.030,-39.020,-179.693,5.241,148.813
C04297=1236.320,-29.781,-39.033,-179.689,5.242,148.813
C04298=1236.315,-29.531,-39.047,-179.687,5.242,148.812
C04299=1236.310,-29.282,-39.060,-179.685,5.242,148.811
C04300=1236.305,-29.031,-39.073,-179.682,5.242,148.810
C04301=1236.300,-28.783,-39.087,-179.680,5.242,148.810
C04302=1236.295,-28.532,-39.100,-179.677,5.243,148.809
C04303=1236.290,-28.284,-39.114,-179.675,5.243,148.808
C04304=1236.285,-28.033,-39.127,-179.672,5.243,148.808
C04305=1236.280,-27.785,-39.141,-179.670,5.243,148.807
C04306=1236.275,-27.534,-39.154,-179.668,5.243,148.806
C04307=1236.269,-27.285,-39.168,-179.665,5.243,148.806
C04308=1236.265,-27.035,-39.181,-179.662,5.244,148.805
C04309=1236.260,-26.786,-39.195,-179.660,5.244,148.804
C04310=1236.255,-26.536,-39.208,-179.658,5.244,148.803
C04311=1236.250,-26.286,-39.222,-179.655,5.244,148.803
C04312=1236.244,-26.037,-39.235,-179.652,5.244,148.802
C04313=1236.240,-25.787,-39.249,-179.650,5.245,148.801
C04314=1236.234,-25.538,-39.262,-179.648,5.244,148.800
C04315=1236.230,-25.288,-39.276,-179.645,5.245,148.800
C04316=1236.224,-25.038,-39.289,-179.643,5.244,148.799
C04317=1236.219,-24.789,-39.303,-179.640,5.245,148.798
C04318=1236.214,-24.539,-39.316,-179.638,5.245,148.798
C04319=1236.209,-24.290,-39.330,-179.636,5.245,148.797
C04320=1236.204,-24.041,-39.344,-179.633,5.246,148.796
C04321=1236.199,-23.790,-39.358,-179.630,5.246,148.796
C04322=1236.194,-23.541,-39.371,-179.628,5.246,148.795
C04323=1236.189,-23.291,-39.384,-179.625,5.246,148.794
C04324=1236.184,-23.042,-39.398,-179.623,5.246,148.793
C04325=1236.179,-22.793,-39.413,-179.621,5.247,148.793
C04326=1236.173,-22.523,-39.428,-179.618,5.247,148.792
C04327=1236.168,-22.254,-39.442,-179.615,5.247,148.791
C04328=1236.162,-21.985,-39.457,-179.613,5.247,148.790
C04329=1236.157,-21.715,-39.471,-179.610,5.247,148.790
C04330=1236.152,-21.466,-39.485,-179.607,5.248,148.789
C04331=1236.146,-21.217,-39.499,-179.605,5.247,148.788
C04332=1236.142,-20.967,-39.512,-179.602,5.248,148.787
C04333=1236.137,-20.717,-39.526,-179.600,5.248,148.787
C04334=1236.131,-20.468,-39.540,-179.598,5.248,148.786
C04335=1236.127,-20.218,-39.554,-179.595,5.249,148.785
C04336=1236.122,-19.968,-39.567,-179.593,5.248,148.785
C04337=1236.116,-19.719,-39.581,-179.590,5.249,148.784
C04338=1236.111,-19.469,-39.596,-179.587,5.249,148.783
C04339=1236.107,-19.219,-39.609,-179.585,5.249,148.783
C04340=1236.101,-18.970,-39.623,-179.583,5.250,148.782
C04341=1236.096,-18.721,-39.637,-179.580,5.250,148.781
C04342=1236.091,-18.471,-39.651,-179.578,5.249,148.780
C04343=1236.086,-18.222,-39.664,-179.575,5.250,148.780
C04344=1236.081,-17.972,-39.678,-179.573,5.250,148.779
C04345=1236.076,-17.722,-39.692,-179.570,5.250,148.778
C04346=1236.071,-17.473,-39.706,-179.567,5.251,148.778
C04347=1236.065,-17.223,-39.720,-179.565,5.250,148.777
C04348=1236.061,-16.973,-39.733,-179.563,5.251,148.776
C04349=1236.056,-16.724,-39.747,-179.560,5.251,148.775
C04350=1236.051,-16.475,-39.762,-179.558,5.251,148.775
C04351=1236.046,-16.225,-39.776,-179.555,5.252,148.774
C04352=1236.040,-15.975,-39.789,-179.553,5.252,148.773
C04353=1236.036,-15.726,-39.803,-179.551,5.252,148.773
C04354=1236.031,-15.476,-39.817,-179.548,5.252,148.772
C04355=1236.026,-15.227,-39.831,-179.546,5.252,148.771
C04356=1236.020,-14.978,-39.845,-179.543,5.253,148.771
C04357=1236.015,-14.728,-39.859,-179.540,5.253,148.770
C04358=1236.010,-14.478,-39.874,-179.538,5.253,148.769
C04359=1236.005,-14.228,-39.887,-179.535,5.253,148.768
C04360=1236.000,-13.979,-39.901,-179.533,5.254,148.768
C04361=1235.995,-13.729,-39.915,-179.531,5.253,148.767
C04362=1235.990,-13.480,-39.929,-179.528,5.254,148.766
C04363=1235.985,-13.230,-39.943,-179.525,5.254,148.765
C04364=1235.980,-12.981,-39.957,-179.523,5.254,148.765
C04365=1235.975,-12.731,-39.972,-179.521,5.255,148.764
C04366=1235.970,-12.482,-39.986,-179.518,5.255,148.763
C04367=1235.965,-12.232,-40.000,-179.516,5.255,148.763
C04368=1235.960,-11.983,-40.014,-179.513,5.255,148.762
C04369=1235.955,-11.733,-40.028,-179.510,5.256,148.761
C04370=1235.950,-11.484,-40.042,-179.508,5.256,148.761
C04371=1235.945,-11.234,-40.056,-179.506,5.256,148.760
C04372=1235.940,-10.985,-40.070,-179.503,5.257,148.759
C04373=1235.935,-10.735,-40.085,-179.500,5.256,148.758
C04374=1235.930,-10.486,-40.099,-179.498,5.256,148.758
C04375=1235.925,-10.236,-40.113,-179.495,5.257,148.757
C04376=1235.920,-9.986,-40.127,-179.493,5.257,148.756
C04377=1235.914,-9.737,-40.141,-179.490,5.257,148.756
C04378=1235.909,-9.487,-40.156,-179.488,5.257,148.755
C04379=1235.904,-9.238,-40.170,-179.486,5.257,148.754
C04380=1235.899,-8.988,-40.184,-179.483,5.258,148.753
C04381=1235.894,-8.738,-40.198,-179.481,5.258,148.753
C04382=1235.889,-8.489,-40.212,-179.478,5.258,148.752
C04383=1235.884,-8.240,-40.227,-179.476,5.259,148.751
C04384=1235.879,-7.990,-40.241,-179.474,5.258,148.751
C04385=1235.874,-7.740,-40.255,-179.471,5.259,148.750
C04386=1235.869,-7.490,-40.269,-179.468,5.259,148.749
C04387=1235.864,-7.241,-40.284,-179.466,5.259,148.749
C04388=1235.858,-6.992,-40.298,-179.464,5.260,148.748
C04389=1235.854,-6.742,-40.312,-179.461,5.260,148.747
C04390=1235.849,-6.492,-40.326,-179.459,5.260,148.747
C04391=1235.844,-6.243,-40.340,-179.456,5.261,148.746
C04392=1235.839,-5.994,-40.355,-179.453,5.261,148.745
C04393=1235.834,-5.744,-40.370,-179.451,5.260,148.744
C04394=1235.829,-5.494,-40.384,-179.448,5.261,148.744
C04395=1235.824,-5.245,-40.398,-179.446,5.261,148.743
C04396=1235.819,-4.995,-40.412,-179.443,5.262,148.742
C04397=1235.814,-4.746,-40.426,-179.441,5.262,148.741
C04398=1235.809,-4.497,-40.441,-179.438,5.262,148.741
C04399=1235.804,-4.247,-40.456,-179.436,5.263,148.740
C04400=1235.799,-3.997,-40.470,-179.433,5.262,148.739
C04401=1235.794,-3.747,-40.484,-179.431,5.263,148.739
C04402=1235.789,-3.498,-40.499,-179.428,5.264,148.738
C04403=1235.784,-3.249,-40.512,-179.426,5.263,148.737
C04404=1235.778,-2.999,-40.528,-179.423,5.264,148.737
C04405=1235.773,-2.750,-40.542,-179.421,5.264,148.736
C04406=1235.768,-2.500,-40.557,-179.419,5.264,148.735
C04407=1235.763,-2.250,-40.571,-179.416,5.265,148.735
C04408=1235.759,-2.001,-40.586,-179.413,5.265,148.734
C04409=1235.754,-1.751,-40.600,-179.411,5.265,148.733
C04410=1235.749,-1.502,-40.614,-179.409,5.265,148.733
C04411=1235.744,-1.252,-40.629,-179.406,5.266,148.732
C04412=1235.739,-1.003,-40.644,-179.403,5.265,148.731
C04413=1235.733,-0.753,-40.659,-179.401,5.266,148.730
C04414=1235.728,-0.504,-40.672,-179.398,5.266,148.730
C04415=1235.723,-0.255,-40.687,-179.396,5.266,148.729
C04416=1235.718,-0.005,-40.702,-179.393,5.267,148.728
C04417=1235.713,0.245,-40.716,-179.391,5.267,148.727
C04418=1235.709,0.494,-40.731,-179.388,5.268,148.727
C04419=1235.703,0.744,-40.746,-179.386,5.267,148.726
C04420=1235.698,0.993,-40.760,-179.383,5.268,148.725
C04421=1235.693,1.243,-40.775,-179.381,5.268,148.725
C04422=1235.688,1.492,-40.789,-179.379,5.268,148.724
C04423=1235.683,1.742,-40.804,-179.376,5.269,148.723
C04424=1235.678,1.991,-40.819,-179.373,5.269,148.723
C04425=1235.673,2.241,-40.834,-179.371,5.269,148.722
C04426=1235.668,2.491,-40.848,-179.369,5.269,148.721
C04427=1235.664,2.740,-40.863,-179.366,5.270,148.721
C04428=1235.658,2.990,-40.878,-179.363,5.271,148.720
C04429=1235.653,3.239,-40.893,-179.361,5.270,148.719
C04430=1235.648,3.508,-40.908,-179.359,5.271,148.718
C04431=1235.643,3.777,-40.924,-179.355,5.271,148.718
C04432=1235.637,4.046,-40.940,-179.353,5.271,148.717
C04433=1235.632,4.314,-40.956,-179.350,5.272,148.716
C04434=1235.627,4.564,-40.970,-179.348,5.272,148.716
C04435=1235.621,4.814,-40.985,-179.345,5.272,148.715
C04436=1235.617,5.063,-41.000,-179.343,5.273,148.714
C04437=1235.612,5.313,-41.015,-179.341,5.273,148.713
C04438=1235.607,5.562,-41.030,-179.338,5.273,148.713
C04439=1235.601,5.812,-41.044,-179.335,5.274,148.712
C04440=1235.597,6.061,-41.059,-179.332,5.274,148.711
C04441=1235.592,6.311,-41.074,-179.330,5.274,148.710
C04442=1235.586,6.560,-41.089,-179.327,5.274,148.710
C04443=1235.581,6.810,-41.104,-179.325,5.275,148.709
C04444=1235.577,7.059,-41.119,-179.323,5.274,148.708
C04445=1235.571,7.309,-41.133,-179.320,5.275,148.708
C04446=1235.566,7.558,-41.148,-179.317,5.275,148.707
C04447=1235.562,7.807,-41.163,-179.315,5.276,148.706
C04448=1235.556,8.057,-41.178,-179.313,5.276,148.706
C04449=1235.551,8.306,-41.193,-179.310,5.276,148.705
C04450=1235.546,8.556,-41.208,-179.307,5.277,148.704
C04451=1235.541,8.806,-41.223,-179.305,5.276,148.704
C04452=1235.536,9.055,-41.237,-179.303,5.277,148.703
C04453=1235.532,9.304,-41.252,-179.300,5.278,148.702
C04454=1235.526,9.554,-41.268,-179.297,5.278,148.702
C04455=1235.521,9.803,-41.282,-179.295,5.278,148.701
C04456=1235.517,10.053,-41.297,-179.293,5.278,148.700
C04457=1235.511,10.303,-41.313,-179.290,5.279,148.699
C04458=1235.507,10.552,-41.328,-179.288,5.279,148.699
C04459=1235.501,10.802,-41.343,-179.285,5.279,148.698
C04460=1235.496,11.052,-41.357,-179.283,5.280,148.697
C04461=1235.492,11.301,-41.372,-179.280,5.280,148.697
C04462=1235.486,11.550,-41.388,-179.278,5.280,148.696
C04463=1235.481,11.800,-41.402,-179.275,5.281,148.695
C04464=1235.476,12.049,-41.418,-179.273,5.281,148.695
C04465=1235.471,12.298,-41.433,-179.270,5.282,148.694
C04466=1235.466,12.548,-41.448,-179.268,5.281,148.693
C04467=1235.462,12.798,-41.463,-179.265,5.282,148.693
C04468=1235.457,13.047,-41.478,-179.263,5.282,148.692
C04469=1235.452,13.297,-41.494,-179.260,5.283,148.691
C04470=1235.447,13.546,-41.508,-179.258,5.283,148.691
C04471=1235.441,13.796,-41.523,-179.255,5.283,148.690
C04472=1235.437,14.045,-41.538,-179.253,5.284,148.689
C04473=1235.431,14.294,-41.554,-179.250,5.284,148.689
C04474=1235.426,14.544,-41.568,-179.248,5.284,148.688
C04475=1235.422,14.794,-41.584,-179.245,5.285,148.687
C04476=1235.417,15.043,-41.599,-179.243,5.285,148.686
C04477=1235.411,15.292,-41.615,-179.240,5.285,148.686
C04478=1235.407,15.542,-41.629,-179.238,5.285,148.685
C04479=1235.401,15.792,-41.645,-179.235,5.286,148.684
C04480=1235.396,16.041,-41.660,-179.233,5.287,148.684
C04481=1235.392,16.291,-41.676,-179.230,5.286,148.683
C04482=1235.387,16.540,-41.691,-179.228,5.287,148.682
C04483=1235.381,16.790,-41.706,-179.225,5.287,148.682
C04484=1235.377,17.039,-41.721,-179.223,5.288,148.681
C04485=1235.371,17.288,-41.736,-179.220,5.287,148.680
C04486=1235.367,17.537,-41.751,-179.217,5.288,148.679
C04487=1235.362,17.788,-41.767,-179.215,5.288,148.679
C04488=1235.356,18.037,-41.783,-179.212,5.289,148.678
C04489=1235.352,18.286,-41.798,-179.210,5.289,148.677
C04490=1235.346,18.536,-41.813,-179.207,5.289,148.677
C04491=1235.342,18.785,-41.828,-179.205,5.290,148.676
C04492=1235.337,19.035,-41.843,-179.202,5.290,148.675
C04493=1235.332,19.284,-41.858,-179.200,5.290,148.675
C04494=1235.327,19.534,-41.874,-179.197,5.291,148.674
C04495=1235.321,19.783,-41.890,-179.195,5.291,148.673
C04496=1235.317,20.033,-41.905,-179.192,5.292,148.673
C04497=1235.312,20.282,-41.921,-179.189,5.292,148.672
C04498=1235.307,20.531,-41.936,-179.187,5.292,148.671
C04499=1235.302,20.781,-41.951,-179.185,5.293,148.671
C04500=1235.296,21.030,-41.967,-179.182,5.293,148.670
C04501=1235.292,21.280,-41.982,-179.179,5.294,148.669
C04502=1235.287,21.529,-41.998,-179.177,5.293,148.668
C04503=1235.282,21.779,-42.013,-179.175,5.294,148.668
C04504=1235.277,22.028,-42.028,-179.172,5.294,148.667
C04505=1235.272,22.278,-42.044,-179.169,5.295,148.666
C04506=1235.267,22.527,-42.060,-179.167,5.295,148.666
C04507=1235.262,22.777,-42.075,-179.165,5.295,148.665
C04508=1235.257,23.026,-42.090,-179.162,5.296,148.664
C04509=1235.252,23.276,-42.106,-179.159,5.296,148.664
C04510=1235.247,23.525,-42.121,-179.157,5.297,148.663
C04511=1235.242,23.775,-42.137,-179.155,5.297,148.662
C04512=1235.237,24.025,-42.153,-179.152,5.297,148.662
C04513=1235.233,24.274,-42.168,-179.149,5.298,148.661
C04514=1235.227,24.523,-42.183,-179.147,5.298,148.660
C04515=1235.222,24.773,-42.199,-179.145,5.298,148.660
C04516=1235.218,25.022,-42.214,-179.142,5.299,148.659
C04517=1235.212,25.272,-42.230,-179.139,5.299,148.658
C04518=1235.207,25.521,-42.246,-179.137,5.300,148.658
C04519=1235.202,25.771,-42.262,-179.134,5.300,148.657
C04520=1235.198,26.020,-42.277,-179.132,5.300,148.656
C04521=1235.192,26.269,-42.293,-179.130,5.301,148.656
C04522=1235.188,26.519,-42.309,-179.127,5.302,148.655
C04523=1235.182,26.769,-42.324,-179.124,5.302,148.654
C04524=1235.178,27.018,-42.339,-179.122,5.302,148.654
C04525=1235.173,27.268,-42.355,-179.120,5.302,148.653
C04526=1235.168,27.517,-42.372,-179.117,5.303,148.652
C04527=1235.162,27.766,-42.387,-179.114,5.304,148.652
C04528=1235.158,28.016,-42.403,-179.112,5.304,148.651
C04529=1235.153,28.265,-42.418,-179.110,5.304,148.650
C04530=1235.147,28.515,-42.434,-179.107,5.304,148.650
C04531=1235.143,28.764,-42.450,-179.104,5.305,148.649
C04532=1235.138,29.013,-42.466,-179.102,5.305,148.648
C04533=1235.133,29.263,-42.481,-179.099,5.306,148.648
C04534=1235.127,29.531,-42.498,-179.096,5.306,148.647
C04535=1235.122,29.800,-42.515,-179.094,5.306,148.646
C04536=1235.117,30.069,-42.532,-179.091,5.307,148.645
C04537=1235.111,30.337,-42.549,-179.089,5.307,148.645
C04538=1235.106,30.587,-42.565,-179.086,5.308,148.644
C04539=1235.101,30.837,-42.581,-179.083,5.308,148.643
C04540=1235.097,31.085,-42.597,-179.081,5.309,148.643
C04541=1235.092,31.335,-42.613,-179.078,5.309,148.642
C04542=1235.087,31.585,-42.628,-179.076,5.309,148.641
C04543=1235.082,31.833,-42.645,-179.073,5.310,148.641
C04544=1235.077,32.084,-42.660,-179.071,5.310,148.640
C04545=1235.071,32.333,-42.676,-179.068,5.311,148.639
C04546=1235.067,32.582,-42.693,-179.065,5.311,148.639
C04547=1235.062,32.832,-42.708,-179.063,5.311,148.638
C04548=1235.057,33.081,-42.723,-179.061,5.312,148.637
C04549=1235.052,33.330,-42.740,-179.058,5.312,148.637
C04550=1235.047,33.580,-42.756,-179.055,5.313,148.636
C04551=1235.042,33.830,-42.772,-179.053,5.313,148.635
C04552=1235.037,34.079,-42.788,-179.051,5.313,148.634
C04553=1235.032,34.329,-42.804,-179.048,5.314,148.634
C04554=1235.027,34.578,-42.820,-179.045,5.314,148.633
C04555=1235.022,34.827,-42.836,-179.043,5.315,148.632
C04556=1235.017,35.077,-42.852,-179.040,5.315,148.632
C04557=1235.012,35.326,-42.868,-179.038,5.316,148.631
C04558=1235.007,35.576,-42.884,-179.035,5.316,148.630
C04559=1235.002,35.825,-42.900,-179.033,5.317,148.630
C04560=1234.997,36.075,-42.916,-179.031,5.317,148.629
C04561=1234.992,36.324,-42.932,-179.028,5.318,148.629
C04562=1234.988,36.574,-42.948,-179.025,5.318,148.628
C04563=1234.983,36.823,-42.963,-179.023,5.319,148.627
C04564=1234.978,37.072,-42.980,-179.021,5.319,148.627
C04565=1234.973,37.322,-42.996,-179.018,5.319,148.626
C04566=1234.968,37.571,-43.012,-179.015,5.320,148.625
C04567=1234.963,37.821,-43.028,-179.013,5.320,148.625
C04568=1234.958,38.069,-43.044,-179.010,5.321,148.624
C04569=1234.953,38.320,-43.061,-179.008,5.321,148.623
C04570=1234.947,38.569,-43.077,-179.005,5.321,148.623
C04571=1234.943,38.819,-43.093,-179.003,5.322,148.622
C04572=1234.938,39.067,-43.109,-179.000,5.322,148.621
C04573=1234.933,39.317,-43.126,-178.997,5.323,148.621
C04574=1234.928,39.566,-43.142,-178.995,5.323,148.620
C04575=1234.923,39.816,-43.158,-178.992,5.324,148.619
C04576=1234.918,40.065,-43.174,-178.990,5.324,148.618
C04577=1234.913,40.315,-43.191,-178.987,5.324,148.618
C04578=1234.908,40.564,-43.206,-178.985,5.325,148.617
C04579=1234.904,40.814,-43.223,-178.982,5.325,148.616
C04580=1234.898,41.062,-43.239,-178.980,5.326,148.616
C04581=1234.894,41.313,-43.255,-178.977,5.327,148.615
C04582=1234.889,41.561,-43.271,-178.975,5.327,148.615
C04583=1234.884,41.811,-43.287,-178.973,5.327,148.614
C04584=1234.879,42.061,-43.304,-178.970,5.328,148.613
C04585=1234.873,42.310,-43.321,-178.967,5.328,148.613
C04586=1234.869,42.560,-43.337,-178.965,5.329,148.612
C04587=1234.864,42.809,-43.353,-178.962,5.330,148.611
C04588=1234.859,43.058,-43.370,-178.959,5.330,148.611
C04589=1234.854,43.308,-43.385,-178.957,5.330,148.610
C04590=1234.849,43.557,-43.402,-178.955,5.330,148.609
C04591=1234.844,43.806,-43.418,-178.952,5.331,148.609
C04592=1234.840,44.055,-43.435,-178.950,5.332,148.608
C04593=1234.834,44.306,-43.452,-178.947,5.332,148.607
C04594=1234.829,44.555,-43.468,-178.944,5.333,148.607
C04595=1234.825,44.804,-43.485,-178.942,5.333,148.606
C04596=1234.819,45.054,-43.500,-178.940,5.333,148.605
C04597=1234.815,45.303,-43.517,-178.937,5.334,148.605
C04598=1234.810,45.553,-43.533,-178.935,5.335,148.604
C04599=1234.804,45.802,-43.550,-178.932,5.335,148.603
C04600=1234.800,46.052,-43.566,-178.929,5.336,148.603
C04601=1234.795,46.301,-43.583,-178.927,5.336,148.602
C04602=1234.790,46.550,-43.599,-178.924,5.337,148.601
C04603=1234.786,46.799,-43.616,-178.922,5.337,148.601
C04604=1234.780,47.049,-43.633,-178.919,5.337,148.600
C04605=1234.775,47.299,-43.649,-178.917,5.338,148.599
C04606=1234.770,47.547,-43.665,-178.914,5.338,148.599
C04607=1234.765,47.797,-43.682,-178.912,5.339,148.598
C04608=1234.760,48.047,-43.699,-178.909,5.339,148.597
C04609=1234.755,48.296,-43.715,-178.906,5.340,148.597
C04610=1234.751,48.545,-43.732,-178.904,5.341,148.596
C04611=1234.746,48.795,-43.748,-178.902,5.341,148.596
C04612=1234.740,49.044,-43.765,-178.899,5.341,148.595
C04613=1234.736,49.294,-43.782,-178.897,5.342,148.594
C04614=1234.731,49.543,-43.798,-178.894,5.342,148.594
C04615=1234.726,49.792,-43.815,-178.892,5.343,148.593
C04616=1234.721,50.042,-43.832,-178.889,5.344,148.592
C04617=1234.716,50.291,-43.848,-178.886,5.344,148.592
C04618=1234.711,50.540,-43.865,-178.884,5.345,148.591
C04619=1234.707,50.790,-43.881,-178.882,5.344,148.590
C04620=1234.701,51.040,-43.898,-178.879,5.345,148.590
C04621=1234.696,51.289,-43.914,-178.876,5.346,148.589
C04622=1234.692,51.538,-43.931,-178.874,5.346,148.588
C04623=1234.686,51.788,-43.948,-178.871,5.347,148.588
C04624=1234.681,52.037,-43.965,-178.869,5.348,148.587
C04625=1234.677,52.286,-43.981,-178.866,5.348,148.586
C04626=1234.672,52.536,-43.998,-178.864,5.349,148.586
C04627=1234.667,52.785,-44.015,-178.861,5.349,148.585
C04628=1234.662,53.034,-44.031,-178.859,5.349,148.584
C04629=1234.657,53.284,-44.049,-178.856,5.350,148.584
C04630=1234.652,53.534,-44.065,-178.854,5.350,148.583
C04631=1234.647,53.782,-44.082,-178.851,5.351,148.582
C04632=1234.642,54.032,-44.099,-178.848,5.352,148.582
C04633=1234.638,54.282,-44.116,-178.846,5.352,148.581
C04634=1234.632,54.531,-44.132,-178.844,5.353,148.581
C04635=1234.627,54.780,-44.149,-178.841,5.354,148.580
C04636=1234.623,55.029,-44.167,-178.838,5.354,148.579
C04637=1234.618,55.279,-44.184,-178.836,5.355,148.579
C04638=1234.613,55.547,-44.202,-178.833,5.355,148.578
C04639=1234.607,55.816,-44.220,-178.830,5.356,148.577
C04640=1234.602,56.084,-44.237,-178.827,5.356,148.576
C04641=1234.596,56.353,-44.256,-178.825,5.357,148.576
C04642=1234.592,56.602,-44.273,-178.822,5.357,148.575
C04643=1234.586,56.851,-44.290,-178.820,5.358,148.575
C04644=1234.582,57.100,-44.307,-178.817,5.359,148.574
C04645=1234.577,57.350,-44.324,-178.815,5.359,148.573
C04646=1234.572,57.600,-44.341,-178.813,5.359,148.573
C04647=1234.567,57.848,-44.357,-178.810,5.360,148.572
C04648=1234.562,58.098,-44.374,-178.807,5.360,148.571
C04649=1234.558,58.347,-44.392,-178.805,5.361,148.571
C04650=1234.553,58.597,-44.409,-178.802,5.362,148.570
C04651=1234.548,58.846,-44.426,-178.799,5.362,148.569
C04652=1234.542,59.096,-44.443,-178.797,5.363,148.569
C04653=1234.538,59.345,-44.459,-178.795,5.364,148.568
C04654=1234.533,59.594,-44.477,-178.792,5.364,148.568
C04655=1234.528,59.844,-44.494,-178.789,5.365,148.567
C04656=1234.523,60.093,-44.511,-178.787,5.365,148.566
C04657=1234.518,60.342,-44.527,-178.784,5.366,148.566
C04658=1234.513,60.592,-44.545,-178.782,5.366,148.565
C04659=1234.509,60.841,-44.562,-178.779,5.366,148.564
C04660=1234.503,61.091,-44.579,-178.777,5.367,148.564
C04661=1234.499,61.340,-44.596,-178.775,5.368,148.563
C04662=1234.494,61.589,-44.614,-178.772,5.368,148.562
C04663=1234.488,61.838,-44.631,-178.769,5.369,148.562
C04664=1234.484,62.088,-44.648,-178.767,5.370,148.561
C04665=1234.479,62.338,-44.665,-178.764,5.370,148.560
C04666=1234.474,62.587,-44.682,-178.761,5.371,148.560
C04667=1234.469,62.836,-44.700,-178.759,5.371,148.559
C04668=1234.465,63.086,-44.716,-178.756,5.372,148.558
C04669=1234.460,63.335,-44.734,-178.754,5.373,148.558
C04670=1234.454,63.584,-44.751,-178.751,5.374,148.557
C04671=1234.449,63.834,-44.768,-178.749,5.374,148.557
C04672=1234.445,64.083,-44.786,-178.746,5.375,148.556
C04673=1234.440,64.332,-44.802,-178.743,5.375,148.555
C04674=1234.435,64.581,-44.820,-178.741,5.375,148.555
C04675=1234.430,64.831,-44.838,-178.739,5.376,148.554
C04676=1234.425,65.081,-44.854,-178.737,5.377,148.554
C04677=1234.421,65.330,-44.872,-178.734,5.377,148.553
C04678=1234.415,65.579,-44.889,-178.731,5.378,148.552
C04679=1234.411,65.828,-44.907,-178.729,5.378,148.552
C04680=1234.405,66.078,-44.924,-178.726,5.379,148.551
C04681=1234.400,66.327,-44.941,-178.724,5.380,148.550
C04682=1234.396,66.576,-44.958,-178.721,5.380,148.550
C04683=1234.391,66.826,-44.976,-178.718,5.381,148.549
C04684=1234.386,67.075,-44.994,-178.716,5.382,148.549
C04685=1234.381,67.325,-45.010,-178.713,5.382,148.548
C04686=1234.376,67.574,-45.028,-178.711,5.383,148.547
C04687=1234.371,67.824,-45.046,-178.708,5.383,148.547
C04688=1234.367,68.073,-45.063,-178.706,5.384,148.546
C04689=1234.362,68.322,-45.080,-178.703,5.385,148.545
C04690=1234.357,68.572,-45.098,-178.701,5.386,148.545
C04691=1234.352,68.820,-45.115,-178.698,5.386,148.544
C04692=1234.347,69.070,-45.133,-178.696,5.387,148.543
C04693=1234.342,69.319,-45.150,-178.693,5.387,148.543
C04694=1234.337,69.569,-45.168,-178.690,5.388,148.542
C04695=1234.333,69.817,-45.185,-178.688,5.388,148.541
C04696=1234.327,70.067,-45.202,-178.685,5.389,148.541
C04697=1234.322,70.316,-45.220,-178.683,5.390,148.540
C04698=1234.317,70.566,-45.238,-178.680,5.391,148.540
C04699=1234.313,70.815,-45.255,-178.678,5.391,148.539
C04700=1234.308,71.065,-45.272,-178.676,5.391,148.538
C04701=1234.303,71.314,-45.290,-178.673,5.392,148.538
C04702=1234.298,71.563,-45.308,-178.670,5.392,148.537
C04703=1234.294,71.813,-45.325,-178.668,5.393,148.537
C04704=1234.289,72.062,-45.343,-178.666,5.394,148.536
C04705=1234.284,72.311,-45.361,-178.663,5.394,148.535
C04706=1234.278,72.561,-45.378,-178.660,5.395,148.535
C04707=1234.274,72.810,-45.396,-178.658,5.396,148.534
C04708=1234.269,73.059,-45.414,-178.655,5.396,148.533
C04709=1234.264,73.309,-45.431,-178.653,5.397,148.533
C04710=1234.259,73.558,-45.449,-178.650,5.398,148.532
C04711=1234.254,73.807,-45.467,-178.648,5.398,148.532
C04712=1234.249,74.057,-45.484,-178.645,5.399,148.531
C04713=1234.244,74.306,-45.502,-178.642,5.399,148.530
C04714=1234.239,74.555,-45.520,-178.640,5.400,148.530
C04715=1234.235,74.804,-45.537,-178.638,5.401,148.529
C04716=1234.230,75.054,-45.555,-178.635,5.402,148.529
C04717=1234.225,75.303,-45.573,-178.632,5.402,148.528
C04718=1234.220,75.552,-45.591,-178.630,5.403,148.527
C04719=1234.215,75.802,-45.608,-178.627,5.403,148.527
C04720=1234.210,76.051,-45.626,-178.625,5.404,148.526
C04721=1234.206,76.301,-45.644,-178.622,5.405,148.525
C04722=1234.201,76.550,-45.662,-178.620,5.406,148.525
C04723=1234.197,76.799,-45.680,-178.617,5.406,148.524
C04724=1234.191,77.049,-45.697,-178.614,5.407,148.523
C04725=1234.186,77.298,-45.715,-178.612,5.407,148.523
C04726=1234.182,77.547,-45.733,-178.610,5.408,148.522
C04727=1234.177,77.796,-45.751,-178.607,5.409,148.522
C04728=1234.172,78.046,-45.769,-178.604,5.409,148.521
C04729=1234.167,78.295,-45.787,-178.602,5.410,148.520
C04730=1234.162,78.545,-45.804,-178.599,5.411,148.520
C04731=1234.157,78.794,-45.822,-178.597,5.411,148.519
C04732=1234.152,79.043,-45.840,-178.594,5.412,148.519
C04733=1234.147,79.293,-45.858,-178.592,5.413,148.518
C04734=1234.143,79.542,-45.876,-178.589,5.413,148.517
C04735=1234.138,79.791,-45.894,-178.587,5.414,148.517
C04736=1234.133,80.040,-45.912,-178.584,5.415,148.516
C04737=1234.128,80.289,-45.930,-178.582,5.416,148.516
C04738=1234.123,80.539,-45.948,-178.579,5.416,148.515
C04739=1234.118,80.788,-45.966,-178.576,5.418,148.514
C04740=1234.113,81.038,-45.983,-178.573,5.418,148.514
C04741=1234.108,81.287,-46.001,-178.571,5.419,148.513
C04742=1234.103,81.555,-46.021,-178.568,5.419,148.512
C04743=1234.098,81.823,-46.040,-178.566,5.420,148.512
C04744=1234.093,82.092,-46.060,-178.563,5.421,148.511
C04745=1234.088,82.360,-46.079,-178.560,5.421,148.510
C04746=1234.083,82.610,-46.097,-178.558,5.422,148.510
C04747=1234.078,82.859,-46.116,-178.556,5.423,148.509
C04748=1234.073,83.108,-46.134,-178.553,5.423,148.509
C04749=1234.068,83.357,-46.152,-178.550,5.424,148.508
C04750=1234.063,83.607,-46.170,-178.548,5.425,148.507
C04751=1234.058,83.856,-46.188,-178.545,5.426,148.507
C04752=1234.054,84.106,-46.206,-178.542,5.427,148.506
C04753=1234.049,84.355,-46.224,-178.540,5.428,148.506
C04754=1234.044,84.604,-46.242,-178.537,5.428,148.505
C04755=1234.039,84.853,-46.260,-178.535,5.429,148.505
C04756=1234.034,85.102,-46.278,-178.532,5.430,148.504
C04757=1234.030,85.352,-46.297,-178.530,5.430,148.503
C04758=1234.025,85.601,-46.315,-178.527,5.431,148.503
C04759=1234.019,85.850,-46.334,-178.524,5.432,148.502
C04760=1234.014,86.100,-46.352,-178.522,5.433,148.501
C04761=1234.010,86.349,-46.370,-178.520,5.433,148.501
C04762=1234.005,86.599,-46.388,-178.517,5.434,148.500
C04763=1234.000,86.848,-46.406,-178.514,5.434,148.500
C04764=1233.995,87.097,-46.424,-178.512,5.435,148.499
C04765=1233.991,87.346,-46.442,-178.510,5.436,148.498
C04766=1233.986,87.596,-46.462,-178.507,5.437,148.498
C04767=1233.981,87.845,-46.480,-178.504,5.437,148.497
C04768=1233.976,88.094,-46.498,-178.502,5.438,148.496
C04769=1233.971,88.343,-46.516,-178.500,5.439,148.496
C04770=1233.966,88.592,-46.534,-178.497,5.439,148.495
C04771=1233.961,88.842,-46.553,-178.494,5.441,148.495
C04772=1233.956,89.091,-46.571,-178.491,5.441,148.494
C04773=1233.952,89.340,-46.589,-178.489,5.442,148.494
C04774=1233.947,89.589,-46.607,-178.487,5.443,148.493
C04775=1233.943,89.839,-46.626,-178.484,5.444,148.492
C04776=1233.937,90.088,-46.645,-178.481,5.444,148.492
C04777=1233.932,90.337,-46.663,-178.479,5.445,148.491
C04778=1233.928,90.587,-46.681,-178.477,5.446,148.491
C04779=1233.923,90.836,-46.700,-178.474,5.446,148.490
C04780=1233.918,91.085,-46.718,-178.471,5.447,148.489
C04781=1233.913,91.334,-46.736,-178.469,5.448,148.489
C04782=1233.909,91.584,-46.755,-178.467,5.448,148.488
C04783=1233.904,91.833,-46.773,-178.464,5.449,148.488
C04784=1233.898,92.082,-46.792,-178.461,5.451,148.487
C04785=1233.894,92.332,-46.811,-178.459,5.451,148.487
C04786=1233.889,92.581,-46.829,-178.456,5.452,148.486
C04787=1233.884,92.830,-46.847,-178.453,5.453,148.485
C04788=1233.879,93.080,-46.867,-178.451,5.453,148.485
C04789=1233.875,93.329,-46.885,-178.449,5.454,148.484
C04790=1233.870,93.578,-46.903,-178.446,5.455,148.484
C04791=1233.865,93.827,-46.922,-178.443,5.455,148.483
C04792=1233.860,94.077,-46.940,-178.441,5.456,148.482
C04793=1233.855,94.325,-46.959,-178.439,5.457,148.482
C04794=1233.850,94.575,-46.978,-178.436,5.458,148.481
C04795=1233.845,94.825,-46.996,-178.433,5.458,148.480
C04796=1233.841,95.073,-47.015,-178.430,5.460,148.480
C04797=1233.836,95.323,-47.034,-178.428,5.461,148.479
C04798=1233.831,95.572,-47.052,-178.425,5.461,148.479
C04799=1233.826,95.821,-47.070,-178.423,5.462,148.478
C04800=1233.821,96.071,-47.090,-178.420,5.463,148.477
C04801=1233.817,96.320,-47.108,-178.418,5.464,148.477
C04802=1233.811,96.569,-47.127,-178.415,5.464,148.476
C04803=1233.807,96.819,-47.146,-178.413,5.465,148.476
C04804=1233.802,97.067,-47.164,-178.411,5.466,148.475
C04805=1233.797,97.317,-47.183,-178.408,5.466,148.475
C04806=1233.793,97.566,-47.202,-178.405,5.468,148.474
C04807=1233.787,97.815,-47.220,-178.402,5.468,148.473
C04808=1233.783,98.065,-47.239,-178.400,5.469,148.473
C04809=1233.778,98.314,-47.257,-178.398,5.470,148.472
C04810=1233.773,98.563,-47.277,-178.395,5.471,148.472
C04811=1233.768,98.813,-47.295,-178.392,5.471,148.471
C04812=1233.763,99.061,-47.314,-178.390,5.472,148.471
C04813=1233.759,99.311,-47.333,-178.388,5.473,148.470
C04814=1233.753,99.560,-47.352,-178.384,5.474,148.469
C04815=1233.749,99.809,-47.371,-178.382,5.475,148.469
C04816=1233.744,100.059,-47.390,-178.380,5.476,148.468
C04817=1233.739,100.307,-47.408,-178.377,5.476,148.468
C04818=1233.734,100.558,-47.427,-178.374,5.477,148.467
C04819=1233.730,100.806,-47.446,-178.372,5.478,148.467
C04820=1233.725,101.056,-47.466,-178.370,5.479,148.466
C04821=1233.720,101.305,-47.484,-178.367,5.479,148.465
C04822=1233.715,101.554,-47.503,-178.364,5.481,148.465
C04823=1233.711,101.803,-47.522,-178.362,5.482,148.464
C04824=1233.705,102.053,-47.541,-178.359,5.482,148.464
C04825=1233.701,102.302,-47.560,-178.357,5.483,148.463
C04826=1233.696,102.551,-47.579,-178.354,5.484,148.463
C04827=1233.692,102.800,-47.598,-178.352,5.484,148.462
C04828=1233.686,103.049,-47.617,-178.349,5.485,148.461
C04829=1233.682,103.299,-47.636,-178.347,5.486,148.461
C04830=1233.677,103.548,-47.655,-178.344,5.487,148.460
C04831=1233.672,103.797,-47.673,-178.341,5.488,148.460
C04832=1233.667,104.046,-47.693,-178.339,5.489,148.459
C04833=1233.663,104.296,-47.712,-178.337,5.490,148.458
C04834=1233.658,104.544,-47.731,-178.334,5.490,148.458
C04835=1233.652,104.795,-47.750,-178.332,5.491,148.457
C04836=1233.648,105.043,-47.769,-178.329,5.492,148.457
C04837=1233.643,105.293,-47.788,-178.326,5.493,148.456
C04838=1233.639,105.541,-47.807,-178.323,5.494,148.455
C04839=1233.634,105.791,-47.827,-178.321,5.495,148.455
C04840=1233.628,106.040,-47.845,-178.319,5.496,148.454
C04841=1233.624,106.290,-47.864,-178.316,5.496,148.454
C04842=1233.619,106.538,-47.883,-178.314,5.497,148.453
C04843=1233.614,106.788,-47.903,-178.311,5.499,148.453
C04844=1233.609,107.037,-47.922,-178.308,5.499,148.452
C04845=1233.605,107.286,-47.941,-178.306,5.500,148.452
C04846=1233.599,107.555,-47.961,-178.303,5.501,148.451
C04847=1233.594,107.823,-47.983,-178.301,5.501,148.450
C04848=1233.589,108.092,-48.004,-178.298,5.503,148.450
C04849=1233.584,108.360,-48.024,-178.295,5.504,148.449
C04850=1233.580,108.609,-48.043,-178.292,5.504,148.448
C04851=1233.574,108.858,-48.063,-178.290,5.505,148.448
C04852=1233.570,109.107,-48.082,-178.287,5.507,148.447
C04853=1233.565,109.357,-48.100,-178.284,5.507,148.447
C04854=1233.560,109.606,-48.120,-178.282,5.508,148.446
C04855=1233.555,109.856,-48.140,-178.280,5.509,148.446
C04856=1233.550,110.104,-48.158,-178.277,5.509,148.445
C04857=1233.546,110.354,-48.178,-178.274,5.511,148.445
C04858=1233.540,110.603,-48.197,-178.272,5.512,148.444
C04859=1233.536,110.852,-48.216,-178.269,5.512,148.443
C04860=1233.532,111.102,-48.236,-178.267,5.513,148.443
C04861=1233.526,111.351,-48.255,-178.264,5.514,148.442
C04862=1233.521,111.600,-48.275,-178.262,5.515,148.442
C04863=1233.517,111.849,-48.294,-178.259,5.516,148.441
C04864=1233.512,112.098,-48.313,-178.257,5.517,148.441
C04865=1233.507,112.348,-48.333,-178.254,5.518,148.440
C04866=1233.502,112.597,-48.352,-178.252,5.519,148.440
C04867=1233.498,112.846,-48.373,-178.249,5.519,148.439
C04868=1233.493,113.094,-48.391,-178.247,5.521,148.439
C04869=1233.488,113.344,-48.411,-178.244,5.522,148.438
C04870=1233.484,113.593,-48.431,-178.241,5.522,148.437
C04871=1233.478,113.842,-48.450,-178.239,5.523,148.437
C04872=1233.473,114.092,-48.470,-178.237,5.524,148.436
C04873=1233.469,114.341,-48.489,-178.233,5.525,148.436
C04874=1233.464,114.590,-48.508,-178.231,5.526,148.435
C04875=1233.459,114.840,-48.528,-178.229,5.527,148.435
C04876=1233.455,115.088,-48.548,-178.226,5.528,148.434
C04877=1233.450,115.337,-48.567,-178.224,5.529,148.433
C04878=1233.445,115.587,-48.587,-178.221,5.530,148.433
C04879=1233.441,115.836,-48.606,-178.219,5.531,148.432
C04880=1233.435,116.085,-48.625,-178.216,5.532,148.432
C04881=1233.431,116.335,-48.645,-178.213,5.532,148.431
C04882=1233.426,116.584,-48.665,-178.211,5.533,148.431
C04883=1233.421,116.832,-48.685,-178.208,5.535,148.430
C04884=1233.416,117.082,-48.704,-178.206,5.535,148.430
C04885=1233.411,117.332,-48.724,-178.203,5.536,148.429
C04886=1233.406,117.580,-48.743,-178.201,5.537,148.428
C04887=1233.402,117.829,-48.764,-178.198,5.538,148.428
C04888=1233.397,118.079,-48.783,-178.196,5.539,148.427
C04889=1233.393,118.328,-48.802,-178.193,5.540,148.427
C04890=1233.388,118.576,-48.822,-178.191,5.541,148.426
C04891=1233.383,118.826,-48.842,-178.188,5.542,148.426
C04892=1233.378,119.076,-48.862,-178.185,5.543,148.425
C04893=1233.373,119.324,-48.881,-178.183,5.544,148.425
C04894=1233.369,119.573,-48.901,-178.180,5.545,148.424
C04895=1233.364,119.823,-48.921,-178.178,5.546,148.424
C04896=1233.359,120.073,-48.941,-178.176,5.546,148.423
C04897=1233.354,120.321,-48.961,-178.172,5.548,148.422
C04898=1233.349,120.570,-48.980,-178.170,5.549,148.422
C04899=1233.345,120.820,-49.000,-178.168,5.549,148.421
C04900=1233.340,121.069,-49.020,-178.165,5.550,148.421
C04901=1233.335,121.318,-49.040,-178.162,5.552,148.420
C04902=1233.330,121.567,-49.060,-178.160,5.553,148.420
C04903=1233.326,121.816,-49.080,-178.158,5.554,148.419
C04904=1233.321,122.066,-49.099,-178.155,5.554,148.419
C04905=1233.316,122.314,-49.119,-178.152,5.556,148.418
C04906=1233.311,122.564,-49.139,-178.150,5.557,148.418
C04907=1233.307,122.813,-49.159,-178.147,5.557,148.417
C04908=1233.302,123.062,-49.179,-178.145,5.558,148.417
C04909=1233.297,123.312,-49.199,-178.142,5.560,148.416
C04910=1233.292,123.560,-49.219,-178.139,5.560,148.415
C04911=1233.287,123.810,-49.238,-178.137,5.561,148.415
C04912=1233.283,124.058,-49.259,-178.135,5.562,148.414
C04913=1233.278,124.308,-49.278,-178.132,5.564,148.414
C04914=1233.274,124.557,-49.299,-178.129,5.564,148.413
C04915=1233.268,124.806,-49.319,-178.127,5.565,148.413
C04916=1233.263,125.055,-49.339,-178.125,5.566,148.412
C04917=1233.259,125.305,-49.359,-178.121,5.567,148.412
C04918=1233.254,125.554,-49.379,-178.119,5.568,148.411
C04919=1233.249,125.803,-49.399,-178.117,5.569,148.411
C04920=1233.245,126.052,-49.419,-178.115,5.570,148.410
C04921=1233.240,126.300,-49.439,-178.111,5.572,148.410
C04922=1233.235,126.550,-49.459,-178.109,5.572,148.409
C04923=1233.231,126.799,-49.479,-178.107,5.573,148.408
C04924=1233.225,127.049,-49.499,-178.104,5.574,148.408
C04925=1233.221,127.298,-49.520,-178.101,5.576,148.407
C04926=1233.216,127.547,-49.539,-178.099,5.576,148.407
C04927=1233.212,127.796,-49.560,-178.097,5.577,148.406
C04928=1233.207,128.045,-49.580,-178.094,5.579,148.406
C04929=1233.202,128.294,-49.599,-178.091,5.579,148.405
C04930=1233.197,128.543,-49.620,-178.089,5.580,148.405
C04931=1233.192,128.792,-49.641,-178.086,5.581,148.404
C04932=1233.187,129.042,-49.660,-178.084,5.583,148.404
C04933=1233.183,129.291,-49.681,-178.081,5.583,148.403
C04934=1233.179,129.540,-49.701,-178.079,5.584,148.403
C04935=1233.173,129.790,-49.721,-178.076,5.585,148.402
C04936=1233.169,130.039,-49.742,-178.073,5.586,148.401
C04937=1233.164,130.287,-49.762,-178.071,5.587,148.401
C04938=1233.159,130.536,-49.781,-178.068,5.588,148.400
C04939=1233.154,130.785,-49.802,-178.066,5.590,148.400
C04940=1233.149,131.035,-49.823,-178.063,5.591,148.399
C04941=1233.145,131.284,-49.843,-178.061,5.592,148.399
C04942=1233.140,131.533,-49.863,-178.058,5.592,148.398
C04943=1233.136,131.782,-49.883,-178.056,5.594,148.398
C04944=1233.131,132.031,-49.904,-178.053,5.595,148.397
C04945=1233.126,132.280,-49.924,-178.050,5.595,148.397
C04946=1233.121,132.530,-49.944,-178.048,5.597,148.396
C04947=1233.116,132.779,-49.965,-178.045,5.598,148.396
C04948=1233.112,133.028,-49.985,-178.043,5.599,148.395
C04949=1233.107,133.277,-50.006,-178.040,5.600,148.395
C04950=1233.102,133.546,-50.027,-178.037,5.601,148.394
C04951=1233.096,133.814,-50.050,-178.035,5.603,148.394
C04952=1233.092,134.082,-50.072,-178.032,5.603,148.393
C04953=1233.087,134.352,-50.094,-178.029,5.605,148.392
C04954=1233.082,134.601,-50.114,-178.027,5.606,148.392
C04955=1233.077,134.850,-50.135,-178.024,5.606,148.391
C04956=1233.073,135.099,-50.155,-178.022,5.607,148.391
C04957=1233.068,135.347,-50.175,-178.019,5.609,148.390
C04958=1233.062,135.597,-50.196,-178.017,5.610,148.390
C04959=1233.058,135.846,-50.217,-178.014,5.611,148.389
C04960=1233.052,136.096,-50.237,-178.012,5.612,148.389
C04961=1233.048,136.344,-50.257,-178.009,5.613,148.388
C04962=1233.044,136.593,-50.278,-178.006,5.614,148.388
C04963=1233.038,136.843,-50.299,-178.004,5.615,148.387
C04964=1233.034,137.092,-50.319,-178.001,5.616,148.387
C04965=1233.029,137.342,-50.340,-177.999,5.617,148.386
C04966=1233.025,137.591,-50.361,-177.996,5.619,148.386
C04967=1233.021,137.839,-50.381,-177.994,5.620,148.385
C04968=1233.015,138.089,-50.402,-177.991,5.620,148.385
C04969=1233.011,138.338,-50.423,-177.988,5.622,148.384
C04970=1233.006,138.587,-50.443,-177.986,5.623,148.384
C04971=1233.001,138.836,-50.464,-177.984,5.624,148.383
C04972=1232.996,139.085,-50.485,-177.981,5.625,148.383
C04973=1232.992,139.334,-50.505,-177.978,5.626,148.382
C04974=1232.987,139.583,-50.526,-177.976,5.627,148.382
C04975=1232.982,139.832,-50.547,-177.973,5.629,148.381
C04976=1232.978,140.081,-50.568,-177.971,5.629,148.381
C04977=1232.973,140.330,-50.589,-177.968,5.630,148.380
C04978=1232.968,140.579,-50.609,-177.965,5.632,148.380
C04979=1232.963,140.828,-50.630,-177.963,5.633,148.379
C04980=1232.959,141.077,-50.650,-177.961,5.633,148.379
C04981=1232.954,141.326,-50.671,-177.958,5.635,148.378
C04982=1232.949,141.575,-50.692,-177.955,5.636,148.378
C04983=1232.945,141.825,-50.713,-177.953,5.638,148.377
C04984=1232.940,142.074,-50.733,-177.950,5.638,148.377
C04985=1232.935,142.323,-50.755,-177.948,5.639,148.376
C04986=1232.931,142.572,-50.775,-177.945,5.641,148.376
C04987=1232.926,142.821,-50.796,-177.943,5.642,148.375
C04988=1232.920,143.070,-50.817,-177.940,5.642,148.374
C04989=1232.916,143.319,-50.838,-177.937,5.644,148.374
C04990=1232.911,143.568,-50.859,-177.935,5.645,148.373
C04991=1232.907,143.817,-50.880,-177.933,5.646,148.373
C04992=1232.902,144.067,-50.901,-177.930,5.647,148.372
C04993=1232.898,144.316,-50.921,-177.927,5.648,148.372
C04994=1232.892,144.565,-50.942,-177.925,5.649,148.371
C04995=1232.888,144.814,-50.964,-177.922,5.651,148.371
C04996=1232.883,145.063,-50.984,-177.920,5.651,148.370
C04997=1232.878,145.312,-51.005,-177.917,5.653,148.370
C04998=1232.874,145.561,-51.026,-177.914,5.654,148.369
C04999=1232.869,145.810,-51.048,-177.912,5.655,148.369
C05000=1232.864,146.059,-51.069,-177.910,5.657,148.369
C05001=1232.860,146.308,-51.089,-177.907,5.657,148.368
C05002=1232.855,146.557,-51.111,-177.904,5.659,148.368
C05003=1232.850,146.806,-51.132,-177.902,5.660,148.367
C05004=1232.845,147.055,-51.152,-177.900,5.661,148.367
C05005=1232.841,147.305,-51.174,-177.896,5.662,148.366
C05006=1232.836,147.554,-51.195,-177.894,5.663,148.366
C05007=1232.831,147.803,-51.216,-177.892,5.664,148.365
C05008=1232.826,148.051,-51.237,-177.889,5.666,148.365
C05009=1232.821,148.301,-51.258,-177.886,5.666,148.364
C05010=1232.818,148.550,-51.280,-177.884,5.668,148.364
C05011=1232.813,148.799,-51.301,-177.881,5.669,148.363
C05012=1232.807,149.048,-51.322,-177.879,5.670,148.363
C05013=1232.803,149.297,-51.343,-177.876,5.672,148.362
C05014=1232.798,149.546,-51.364,-177.874,5.672,148.362
C05015=1232.794,149.795,-51.386,-177.871,5.674,148.361
C05016=1232.789,150.044,-51.407,-177.869,5.675,148.361
C05017=1232.785,150.293,-51.428,-177.867,5.676,148.360
C05018=1232.779,150.542,-51.449,-177.863,5.677,148.360
C05019=1232.775,150.791,-51.471,-177.861,5.678,148.359
C05020=1232.770,151.041,-51.492,-177.858,5.680,148.359
C05021=1232.766,151.289,-51.513,-177.856,5.681,148.358
C05022=1232.761,151.538,-51.534,-177.853,5.682,148.358
C05023=1232.756,151.787,-51.556,-177.851,5.683,148.357
C05024=1232.751,152.037,-51.577,-177.849,5.684,148.357
C05025=1232.747,152.285,-51.598,-177.845,5.686,148.356
C05026=1232.742,152.534,-51.619,-177.843,5.687,148.356
C05027=1232.738,152.784,-51.641,-177.840,5.688,148.355
C05028=1232.732,153.033,-51.662,-177.838,5.689,148.355
C05029=1232.728,153.282,-51.684,-177.836,5.690,148.354
C05030=1232.722,153.531,-51.705,-177.833,5.692,148.354
C05031=1232.719,153.780,-51.726,-177.831,5.693,148.353
C05032=1232.714,154.029,-51.748,-177.828,5.694,148.353
C05033=1232.709,154.278,-51.769,-177.826,5.695,148.352
C05034=1232.705,154.527,-51.791,-177.823,5.696,148.352
C05035=1232.700,154.776,-51.812,-177.820,5.698,148.352
C05036=1232.694,155.025,-51.833,-177.818,5.698,148.351
C05037=1232.690,155.273,-51.854,-177.815,5.700,148.351
C05038=1232.686,155.523,-51.876,-177.813,5.701,148.350
C05039=1232.681,155.772,-51.897,-177.810,5.703,148.350
C05040=1232.676,156.021,-51.919,-177.808,5.704,148.349
C05041=1232.672,156.270,-51.941,-177.805,5.705,148.349
C05042=1232.667,156.519,-51.962,-177.802,5.706,148.348
C05043=1232.662,156.768,-51.984,-177.800,5.707,148.348
C05044=1232.657,157.017,-52.006,-177.797,5.709,148.347
C05045=1232.652,157.266,-52.027,-177.795,5.710,148.347
C05046=1232.647,157.515,-52.049,-177.792,5.711,148.346
C05047=1232.643,157.764,-52.071,-177.790,5.712,148.346
C05048=1232.639,158.013,-52.092,-177.787,5.714,148.345
C05049=1232.634,158.262,-52.113,-177.785,5.715,148.345
C05050=1232.630,158.511,-52.135,-177.782,5.717,148.344
C05051=1232.625,158.760,-52.156,-177.779,5.717,148.344
C05052=1232.620,159.009,-52.178,-177.777,5.718,148.343
C05053=1232.616,159.258,-52.200,-177.774,5.720,148.343
C05054=1232.610,159.527,-52.223,-177.771,5.722,148.342
C05055=1232.605,159.797,-52.247,-177.769,5.722,148.342
C05056=1232.600,160.065,-52.270,-177.766,5.724,148.341
C05057=1232.595,160.334,-52.294,-177.763,5.726,148.341
C05058=1232.590,160.584,-52.316,-177.761,5.727,148.340
C05059=1232.586,160.832,-52.337,-177.758,5.728,148.340
C05060=1232.581,161.082,-52.359,-177.756,5.729,148.339
C05061=1232.576,161.330,-52.381,-177.754,5.730,148.339
C05062=1232.571,161.580,-52.402,-177.750,5.732,148.339
C05063=1232.567,161.829,-52.424,-177.748,5.733,148.338
C05064=1232.562,162.078,-52.446,-177.745,5.734,148.338
C05065=1232.558,162.327,-52.468,-177.743,5.735,148.337
C05066=1232.553,162.576,-52.490,-177.740,5.737,148.337
C05067=1232.548,162.824,-52.511,-177.738,5.738,148.336
C05068=1232.544,163.074,-52.533,-177.735,5.739,148.336
C05069=1232.539,163.322,-52.555,-177.733,5.740,148.335
C05070=1232.534,163.572,-52.578,-177.730,5.742,148.335
C05071=1232.529,163.821,-52.599,-177.728,5.743,148.334
C05072=1232.525,164.070,-52.621,-177.725,5.744,148.334
C05073=1232.520,164.319,-52.643,-177.723,5.745,148.333
C05074=1232.516,164.568,-52.665,-177.720,5.747,148.333
C05075=1232.511,164.817,-52.687,-177.717,5.748,148.332
C05076=1232.507,165.066,-52.709,-177.715,5.750,148.332
C05077=1232.502,165.315,-52.730,-177.713,5.751,148.332
C05078=1232.497,165.564,-52.753,-177.709,5.752,148.331
C05079=1232.492,165.813,-52.775,-177.707,5.753,148.331
C05080=1232.488,166.062,-52.797,-177.705,5.755,148.330
C05081=1232.483,166.311,-52.819,-177.702,5.756,148.330
C05082=1232.478,166.560,-52.841,-177.699,5.758,148.329
C05083=1232.474,166.808,-52.863,-177.697,5.758,148.329
C05084=1232.470,167.057,-52.885,-177.694,5.760,148.328
C05085=1232.464,167.306,-52.907,-177.692,5.761,148.328
C05086=1232.460,167.556,-52.929,-177.689,5.763,148.327
C05087=1232.455,167.804,-52.951,-177.687,5.764,148.327
C05088=1232.451,168.054,-52.973,-177.684,5.765,148.327
C05089=1232.446,168.302,-52.995,-177.682,5.766,148.326
C05090=1232.441,168.551,-53.018,-177.679,5.768,148.326
C05091=1232.436,168.800,-53.040,-177.677,5.769,148.325
C05092=1232.432,169.049,-53.062,-177.674,5.770,148.325
C05093=1232.427,169.298,-53.084,-177.672,5.771,148.324
C05094=1232.422,169.548,-53.106,-177.669,5.773,148.324
C05095=1232.417,169.796,-53.129,-177.666,5.774,148.323
C05096=1232.413,170.045,-53.151,-177.664,5.776,148.323
C05097=1232.409,170.294,-53.173,-177.662,5.777,148.323
C05098=1232.403,170.543,-53.195,-177.659,5.778,148.322
C05099=1232.399,170.792,-53.218,-177.656,5.779,148.322
C05100=1232.394,171.041,-53.239,-177.654,5.781,148.321
C05101=1232.389,171.290,-53.262,-177.651,5.783,148.321
C05102=1232.385,171.539,-53.284,-177.649,5.784,148.320
C05103=1232.381,171.788,-53.306,-177.646,5.786,148.320
C05104=1232.376,172.037,-53.329,-177.643,5.786,148.319
C05105=1232.371,172.286,-53.351,-177.641,5.788,148.319
C05106=1232.367,172.535,-53.374,-177.639,5.789,148.319
C05107=1232.362,172.783,-53.395,-177.635,5.791,148.318
C05108=1232.357,173.033,-53.418,-177.633,5.792,148.318
C05109=1232.353,173.282,-53.441,-177.631,5.793,148.317
C05110=1232.347,173.531,-53.463,-177.629,5.794,148.317
C05111=1232.343,173.780,-53.485,-177.625,5.796,148.316
C05112=1232.338,174.028,-53.507,-177.623,5.797,148.316
C05113=1232.333,174.278,-53.530,-177.621,5.799,148.316
C05114=1232.330,174.526,-53.553,-177.618,5.800,148.315
C05115=1232.325,174.775,-53.574,-177.616,5.801,148.315
C05116=1232.320,175.025,-53.597,-177.613,5.803,148.314
C05117=1232.316,175.273,-53.620,-177.610,5.804,148.314
C05118=1232.310,175.522,-53.642,-177.608,5.806,148.313
C05119=1232.306,175.771,-53.665,-177.606,5.807,148.313
C05120=1232.302,176.020,-53.687,-177.602,5.808,148.312
C05121=1232.297,176.269,-53.710,-177.600,5.809,148.312
C05122=1232.292,176.518,-53.732,-177.598,5.811,148.312
C05123=1232.288,176.767,-53.755,-177.595,5.813,148.311
C05124=1232.283,177.016,-53.777,-177.592,5.814,148.311
C05125=1232.278,177.265,-53.800,-177.590,5.815,148.310
C05126=1232.274,177.514,-53.822,-177.588,5.816,148.310
C05127=1232.268,177.763,-53.845,-177.585,5.818,148.309
C05128=1232.264,178.012,-53.868,-177.582,5.819,148.309
C05129=1232.259,178.261,-53.891,-177.580,5.821,148.309
C05130=1232.255,178.510,-53.913,-177.577,5.823,148.308
C05131=1232.250,178.759,-53.936,-177.575,5.823,148.308
C05132=1232.246,179.007,-53.959,-177.572,5.825,148.307
C05133=1232.240,179.256,-53.981,-177.570,5.826,148.307
C05134=1232.236,179.505,-54.004,-177.567,5.828,148.306
C05135=1232.231,179.755,-54.026,-177.564,5.829,148.306
C05136=1232.227,180.003,-54.049,-177.562,5.830,148.306
C05137=1232.222,180.252,-54.072,-177.559,5.832,148.305
C05138=1232.218,180.501,-54.094,-177.557,5.833,148.305
C05139=1232.213,180.750,-54.118,-177.554,5.835,148.304
C05140=1232.209,180.999,-54.140,-177.552,5.836,148.304
C05141=1232.204,181.248,-54.163,-177.549,5.838,148.303
C05142=1232.200,181.496,-54.185,-177.546,5.839,148.303
C05143=1232.195,181.745,-54.209,-177.544,5.840,148.303
C05144=1232.190,181.995,-54.231,-177.542,5.842,148.302
C05145=1232.185,182.243,-54.254,-177.539,5.843,148.302
C05146=1232.181,182.492,-54.277,-177.536,5.845,148.301
C05147=1232.177,182.741,-54.300,-177.534,5.846,148.301
C05148=1232.172,182.991,-54.323,-177.532,5.847,148.300
C05149=1232.166,183.239,-54.345,-177.528,5.849,148.300
C05150=1232.162,183.488,-54.368,-177.526,5.851,148.300
C05151=1232.158,183.737,-54.392,-177.524,5.852,148.299
C05152=1232.153,183.986,-54.414,-177.521,5.854,148.299
C05153=1232.149,184.235,-54.437,-177.518,5.854,148.298
C05154=1232.143,184.483,-54.460,-177.516,5.856,148.298
C05155=1232.139,184.732,-54.483,-177.513,5.858,148.297
C05156=1232.135,184.981,-54.506,-177.511,5.859,148.297
C05157=1232.130,185.230,-54.529,-177.508,5.861,148.297
C05158=1232.125,185.500,-54.554,-177.505,5.862,148.296
C05159=1232.120,185.769,-54.579,-177.503,5.864,148.296
C05160=1232.115,186.039,-54.604,-177.500,5.865,148.295
C05161=1232.110,186.309,-54.628,-177.497,5.867,148.295
C05162=1232.106,186.558,-54.652,-177.495,5.869,148.295
C05163=1232.101,186.807,-54.675,-177.492,5.869,148.294
C05164=1232.096,187.056,-54.699,-177.490,5.871,148.294
C05165=1232.092,187.304,-54.721,-177.487,5.873,148.293
C05166=1232.087,187.553,-54.744,-177.485,5.874,148.293
C05167=1232.082,187.802,-54.767,-177.482,5.876,148.292
C05168=1232.077,188.051,-54.790,-177.479,5.877,148.292
C05169=1232.073,188.300,-54.813,-177.477,5.878,148.292
C05170=1232.069,188.549,-54.836,-177.474,5.880,148.291
C05171=1232.064,188.798,-54.860,-177.471,5.882,148.291
C05172=1232.059,189.047,-54.883,-177.469,5.883,148.290
C05173=1232.055,189.295,-54.906,-177.466,5.885,148.290
C05174=1232.050,189.544,-54.929,-177.464,5.887,148.290
C05175=1232.045,189.793,-54.952,-177.462,5.888,148.289
C05176=1232.040,190.042,-54.976,-177.459,5.889,148.289
C05177=1232.036,190.291,-54.999,-177.457,5.890,148.288
C05178=1232.032,190.539,-55.022,-177.454,5.892,148.288
C05179=1232.027,190.789,-55.046,-177.451,5.894,148.288
C05180=1232.023,191.038,-55.069,-177.449,5.895,148.287
C05181=1232.018,191.287,-55.093,-177.446,5.896,148.287
C05182=1232.013,191.536,-55.116,-177.443,5.898,148.286
C05183=1232.008,191.784,-55.139,-177.441,5.899,148.286
C05184=1232.004,192.033,-55.162,-177.439,5.901,148.286
C05185=1231.999,192.282,-55.185,-177.436,5.903,148.285
C05186=1231.995,192.531,-55.208,-177.433,5.904,148.285
C05187=1231.990,192.780,-55.232,-177.431,5.905,148.284
C05188=1231.986,193.028,-55.256,-177.428,5.907,148.284
C05189=1231.981,193.277,-55.279,-177.426,5.908,148.284
C05190=1231.976,193.526,-55.302,-177.423,5.910,148.283
C05191=1231.971,193.775,-55.326,-177.420,5.912,148.283
C05192=1231.967,194.024,-55.349,-177.418,5.913,148.282
C05193=1231.962,194.273,-55.373,-177.416,5.915,148.282
C05194=1231.958,194.521,-55.396,-177.413,5.916,148.282
C05195=1231.954,194.770,-55.419,-177.411,5.917,148.281
C05196=1231.949,195.019,-55.443,-177.408,5.919,148.281
C05197=1231.945,195.268,-55.467,-177.405,5.921,148.280
C05198=1231.940,195.517,-55.490,-177.403,5.923,148.280
C05199=1231.935,195.766,-55.514,-177.400,5.924,148.280
C05200=1231.931,196.015,-55.537,-177.398,5.926,148.279
C05201=1231.926,196.263,-55.561,-177.395,5.927,148.279
C05202=1231.921,196.512,-55.584,-177.393,5.928,148.278
C05203=1231.917,196.761,-55.608,-177.390,5.930,148.278
C05204=1231.912,197.010,-55.632,-177.387,5.932,148.278
C05205=1231.908,197.259,-55.655,-177.385,5.933,148.277
C05206=1231.903,197.508,-55.679,-177.383,5.935,148.277
C05207=1231.899,197.756,-55.703,-177.379,5.936,148.276
C05208=1231.894,198.005,-55.726,-177.377,5.938,148.276
C05209=1231.889,198.254,-55.749,-177.375,5.939,148.276
C05210=1231.885,198.503,-55.773,-177.372,5.941,148.275
C05211=1231.880,198.752,-55.797,-177.369,5.943,148.275
C05212=1231.875,199.001,-55.820,-177.367,5.944,148.274
C05213=1231.871,199.249,-55.844,-177.365,5.946,148.274
C05214=1231.865,199.499,-55.868,-177.362,5.947,148.274
C05215=1231.861,199.747,-55.892,-177.360,5.948,148.273
C05216=1231.856,199.996,-55.916,-177.357,5.950,148.273
C05217=1231.852,200.245,-55.940,-177.354,5.952,148.273
C05218=1231.848,200.494,-55.963,-177.352,5.954,148.272
C05219=1231.844,200.743,-55.987,-177.350,5.955,148.272
C05220=1231.839,200.992,-56.011,-177.346,5.956,148.271
C05221=1231.834,201.240,-56.035,-177.344,5.958,148.271
C05222=1231.830,201.489,-56.058,-177.341,5.960,148.271
C05223=1231.825,201.738,-56.082,-177.339,5.961,148.270
C05224=1231.820,201.987,-56.106,-177.336,5.963,148.270
C05225=1231.815,202.235,-56.130,-177.334,5.965,148.270
C05226=1231.811,202.484,-56.154,-177.332,5.966,148.269
C05227=1231.806,202.733,-56.178,-177.329,5.967,148.269
C05228=1231.802,202.982,-56.201,-177.326,5.969,148.268
C05229=1231.798,203.231,-56.226,-177.323,5.971,148.268
C05230=1231.794,203.479,-56.250,-177.321,5.972,148.268
C05231=1231.788,203.729,-56.274,-177.319,5.974,148.267
C05232=1231.784,203.977,-56.298,-177.316,5.976,148.267
C05233=1231.779,204.226,-56.321,-177.313,5.978,148.267
C05234=1231.775,204.475,-56.345,-177.311,5.979,148.266
C05235=1231.770,204.723,-56.369,-177.308,5.980,148.266
C05236=1231.765,204.973,-56.393,-177.306,5.982,148.265
C05237=1231.761,205.221,-56.418,-177.303,5.984,148.265
C05238=1231.757,205.470,-56.442,-177.301,5.985,148.265
C05239=1231.752,205.719,-56.465,-177.298,5.987,148.264
C05240=1231.747,205.968,-56.490,-177.296,5.989,148.264
C05241=1231.742,206.216,-56.514,-177.293,5.991,148.264
C05242=1231.738,206.466,-56.537,-177.291,5.992,148.263
C05243=1231.734,206.714,-56.562,-177.288,5.993,148.263
C05244=1231.729,206.963,-56.586,-177.285,5.995,148.262
C05245=1231.724,207.211,-56.610,-177.282,5.997,148.262
C05246=1231.720,207.460,-56.634,-177.280,5.998,148.262
C05247=1231.715,207.710,-56.659,-177.278,6.000,148.261
C05248=1231.711,207.958,-56.683,-177.275,6.002,148.261
C05249=1231.706,208.207,-56.707,-177.273,6.004,148.261
C05250=1231.701,208.455,-56.731,-177.270,6.005,148.260
C05251=1231.696,208.704,-56.755,-177.268,6.006,148.260
C05252=1231.693,208.953,-56.779,-177.265,6.008,148.259
C05253=1231.688,209.202,-56.804,-177.262,6.010,148.259
C05254=1231.683,209.451,-56.828,-177.259,6.012,148.259
C05255=1231.679,209.699,-56.852,-177.257,6.013,148.258
C05256=1231.674,209.948,-56.877,-177.255,6.015,148.258
C05257=1231.670,210.197,-56.901,-177.252,6.016,148.258
C05258=1231.665,210.446,-56.925,-177.249,6.018,148.257
C05259=1231.660,210.695,-56.949,-177.247,6.020,148.257
C05260=1231.656,210.944,-56.974,-177.245,6.021,148.257
C05261=1231.651,211.192,-56.998,-177.242,6.023,148.256
C05262=1231.647,211.462,-57.024,-177.239,6.025,148.256
C05263=1231.641,211.733,-57.050,-177.236,6.026,148.255
C05264=1231.637,212.004,-57.078,-177.234,6.028,148.255
C05265=1231.632,212.274,-57.104,-177.231,6.030,148.255
C05266=1231.627,212.522,-57.128,-177.228,6.032,148.254
C05267=1231.622,212.771,-57.153,-177.225,6.034,148.254
C05268=1231.618,213.020,-57.177,-177.223,6.035,148.253
C05269=1231.613,213.269,-57.202,-177.221,6.036,148.253
C05270=1231.609,213.517,-57.226,-177.218,6.038,148.253
C05271=1231.604,213.766,-57.250,-177.215,6.040,148.252
C05272=1231.600,214.015,-57.275,-177.213,6.042,148.252
C05273=1231.595,214.264,-57.299,-177.210,6.044,148.252
C05274=1231.590,214.512,-57.324,-177.208,6.046,148.251
C05275=1231.586,214.762,-57.348,-177.205,6.047,148.251
C05276=1231.581,215.010,-57.373,-177.203,6.049,148.251
C05277=1231.577,215.259,-57.397,-177.200,6.051,148.250
C05278=1231.572,215.508,-57.422,-177.198,6.052,148.250
C05279=1231.568,215.756,-57.447,-177.195,6.054,148.250
C05280=1231.563,216.005,-57.472,-177.193,6.055,148.249
C05281=1231.559,216.254,-57.497,-177.190,6.057,148.249
C05282=1231.554,216.502,-57.521,-177.187,6.059,148.248
C05283=1231.550,216.752,-57.546,-177.185,6.061,148.248
C05284=1231.545,217.000,-57.570,-177.182,6.062,148.248
C05285=1231.540,217.249,-57.595,-177.179,6.064,148.248
C05286=1231.537,217.498,-57.620,-177.177,6.065,148.247
C05287=1231.532,217.746,-57.644,-177.175,6.067,148.247
C05288=1231.527,217.995,-57.669,-177.172,6.069,148.246
C05289=1231.523,218.244,-57.694,-177.169,6.071,148.246
C05290=1231.517,218.493,-57.718,-177.167,6.073,148.246
C05291=1231.514,218.741,-57.743,-177.164,6.075,148.245
C05292=1231.509,218.990,-57.768,-177.162,6.076,148.245
C05293=1231.504,219.239,-57.793,-177.159,6.078,148.245
C05294=1231.500,219.488,-57.817,-177.157,6.079,148.244
C05295=1231.495,219.736,-57.843,-177.154,6.081,148.244
C05296=1231.491,219.985,-57.867,-177.151,6.083,148.244
C05297=1231.486,220.234,-57.892,-177.149,6.085,148.243
C05298=1231.481,220.482,-57.917,-177.147,6.086,148.243
C05299=1231.478,220.731,-57.941,-177.144,6.088,148.243
C05300=1231.472,220.980,-57.966,-177.142,6.090,148.242
C05301=1231.468,221.229,-57.992,-177.139,6.092,148.242
C05302=1231.464,221.477,-58.016,-177.136,6.094,148.242
C05303=1231.459,221.726,-58.041,-177.134,6.095,148.241
C05304=1231.454,221.974,-58.066,-177.132,6.097,148.241
C05305=1231.450,222.224,-58.091,-177.129,6.098,148.241
C05306=1231.446,222.472,-58.116,-177.126,6.100,148.240
C05307=1231.441,222.720,-58.141,-177.124,6.102,148.240
C05308=1231.436,222.970,-58.166,-177.121,6.104,148.240
C05309=1231.432,223.218,-58.191,-177.118,6.106,148.240
C05310=1231.428,223.467,-58.216,-177.116,6.108,148.239
C05311=1231.423,223.715,-58.241,-177.114,6.109,148.239
C05312=1231.418,223.965,-58.266,-177.111,6.111,148.238
C05313=1231.414,224.212,-58.291,-177.109,6.113,148.238
C05314=1231.410,224.462,-58.316,-177.106,6.114,148.238
C05315=1231.405,224.710,-58.341,-177.103,6.116,148.238
C05316=1231.400,224.959,-58.366,-177.101,6.118,148.237
C05317=1231.395,225.207,-58.392,-177.098,6.120,148.237
C05318=1231.392,225.457,-58.416,-177.096,6.121,148.237
C05319=1231.387,225.705,-58.442,-177.093,6.123,148.236
C05320=1231.382,225.954,-58.467,-177.091,6.125,148.236
C05321=1231.377,226.202,-58.492,-177.088,6.127,148.236
C05322=1231.373,226.452,-58.517,-177.085,6.129,148.235
C05323=1231.369,226.699,-58.542,-177.083,6.130,148.235
C05324=1231.364,226.949,-58.567,-177.080,6.132,148.235
C05325=1231.360,227.198,-58.593,-177.078,6.133,148.234
C05326=1231.355,227.446,-58.618,-177.076,6.135,148.234
C05327=1231.351,227.695,-58.643,-177.073,6.137,148.234
C05328=1231.346,227.943,-58.668,-177.070,6.139,148.233
C05329=1231.342,228.192,-58.694,-177.068,6.141,148.233
C05330=1231.337,228.441,-58.719,-177.065,6.143,148.233
C05331=1231.333,228.689,-58.744,-177.062,6.145,148.232
C05332=1231.328,228.937,-58.769,-177.060,6.146,148.232
C05333=1231.324,229.187,-58.794,-177.058,6.147,148.232
C05334=1231.319,229.436,-58.820,-177.055,6.149,148.231
C05335=1231.315,229.684,-58.846,-177.053,6.152,148.231
C05336=1231.310,229.933,-58.871,-177.050,6.153,148.231
C05337=1231.305,230.181,-58.896,-177.048,6.155,148.231
C05338=1231.301,230.430,-58.922,-177.045,6.157,148.230
C05339=1231.297,230.679,-58.948,-177.043,6.159,148.230
C05340=1231.292,230.928,-58.972,-177.040,6.161,148.230
C05341=1231.287,231.176,-58.998,-177.038,6.162,148.229
C05342=1231.283,231.424,-59.023,-177.035,6.164,148.229
C05343=1231.278,231.673,-59.049,-177.033,6.166,148.229
C05344=1231.274,231.923,-59.074,-177.030,6.168,148.228
C05345=1231.269,232.171,-59.099,-177.027,6.169,148.228
C05346=1231.265,232.420,-59.125,-177.025,6.171,148.228
C05347=1231.261,232.668,-59.151,-177.022,6.173,148.227
C05348=1231.256,232.917,-59.176,-177.020,6.175,148.227
C05349=1231.252,233.165,-59.202,-177.017,6.177,148.227
C05350=1231.247,233.414,-59.228,-177.015,6.179,148.227
C05351=1231.242,233.663,-59.253,-177.013,6.180,148.226
C05352=1231.238,233.912,-59.278,-177.010,6.182,148.226
C05353=1231.233,234.160,-59.304,-177.007,6.184,148.226
C05354=1231.229,234.409,-59.329,-177.005,6.186,148.225
C05355=1231.225,234.657,-59.355,-177.002,6.188,148.225
C05356=1231.220,234.906,-59.381,-177.000,6.190,148.225
C05357=1231.216,235.154,-59.406,-176.997,6.191,148.224
C05358=1231.211,235.403,-59.432,-176.994,6.193,148.224
C05359=1231.207,235.652,-59.458,-176.992,6.195,148.224
C05360=1231.202,235.900,-59.483,-176.989,6.197,148.223
C05361=1231.197,236.149,-59.510,-176.988,6.198,148.223
C05362=1231.193,236.398,-59.535,-176.985,6.200,148.223
C05363=1231.188,236.646,-59.561,-176.982,6.202,148.223
C05364=1231.184,236.895,-59.586,-176.980,6.204,148.222
C05365=1231.180,237.144,-59.612,-176.977,6.206,148.222
C05366=1231.175,237.415,-59.640,-176.975,6.208,148.222
C05367=1231.170,237.687,-59.668,-176.972,6.210,148.221
C05368=1231.165,237.957,-59.696,-176.969,6.212,148.221
C05369=1231.160,238.229,-59.724,-176.966,6.214,148.221
C05370=1231.156,238.478,-59.750,-176.963,6.216,148.220
C05371=1231.151,238.727,-59.776,-176.961,6.218,148.220
C05372=1231.146,238.975,-59.802,-176.958,6.220,148.220
C05373=1231.142,239.223,-59.828,-176.956,6.222,148.219
C05374=1231.138,239.472,-59.854,-176.954,6.223,148.219
C05375=1231.134,239.721,-59.880,-176.951,6.225,148.219
C05376=1231.128,239.969,-59.906,-176.949,6.227,148.219
C05377=1231.124,240.218,-59.932,-176.946,6.229,148.218
C05378=1231.120,240.467,-59.957,-176.944,6.231,148.218
C05379=1231.116,240.716,-59.983,-176.941,6.233,148.218
C05380=1231.110,240.964,-60.010,-176.938,6.235,148.217
C05381=1231.106,241.212,-60.035,-176.936,6.236,148.217
C05382=1231.102,241.461,-60.061,-176.934,6.239,148.217
C05383=1231.098,241.710,-60.087,-176.931,6.240,148.217
C05384=1231.093,241.959,-60.114,-176.928,6.242,148.216
C05385=1231.088,242.207,-60.139,-176.926,6.244,148.216
C05386=1231.084,242.455,-60.165,-176.923,6.246,148.216
C05387=1231.079,242.705,-60.192,-176.921,6.248,148.215
C05388=1231.075,242.953,-60.218,-176.918,6.250,148.215
C05389=1231.071,243.202,-60.244,-176.916,6.252,148.215
C05390=1231.067,243.450,-60.269,-176.914,6.253,148.215
C05391=1231.061,243.698,-60.296,-176.911,6.255,148.214
C05392=1231.057,243.947,-60.322,-176.909,6.257,148.214
C05393=1231.053,244.196,-60.348,-176.906,6.259,148.214
C05394=1231.048,244.444,-60.375,-176.904,6.261,148.214
C05395=1231.044,244.693,-60.400,-176.901,6.263,148.213
C05396=1231.039,244.942,-60.427,-176.899,6.265,148.213
C05397=1231.035,245.190,-60.453,-176.896,6.267,148.213
C05398=1231.030,245.438,-60.479,-176.893,6.269,148.212
C05399=1231.025,245.688,-60.505,-176.891,6.270,148.212
C05400=1231.021,245.936,-60.531,-176.889,6.273,148.212
C05401=1231.017,246.185,-60.557,-176.886,6.274,148.212
C05402=1231.013,246.433,-60.584,-176.883,6.276,148.211
C05403=1231.008,246.682,-60.610,-176.881,6.278,148.211
C05404=1231.004,246.930,-60.637,-176.878,6.280,148.211
C05405=1230.999,247.178,-60.662,-176.876,6.282,148.211
C05406=1230.994,247.427,-60.690,-176.873,6.284,148.210
C05407=1230.990,247.676,-60.715,-176.871,6.286,148.210
C05408=1230.986,247.925,-60.741,-176.868,6.288,148.210
C05409=1230.981,248.173,-60.768,-176.866,6.290,148.209
C05410=1230.977,248.421,-60.795,-176.864,6.292,148.209
C05411=1230.972,248.670,-60.821,-176.861,6.294,148.209
C05412=1230.968,248.919,-60.847,-176.858,6.296,148.209
C05413=1230.963,249.168,-60.874,-176.856,6.298,148.208
C05414=1230.959,249.416,-60.900,-176.853,6.300,148.208
C05415=1230.954,249.665,-60.927,-176.851,6.302,148.208
C05416=1230.951,249.913,-60.953,-176.848,6.304,148.208
C05417=1230.946,250.162,-60.979,-176.846,6.306,148.207
C05418=1230.941,250.410,-61.005,-176.843,6.307,148.207
C05419=1230.936,250.658,-61.033,-176.841,6.310,148.207
C05420=1230.932,250.907,-61.058,-176.838,6.312,148.207
C05421=1230.928,251.156,-61.085,-176.836,6.313,148.206
C05422=1230.924,251.404,-61.112,-176.833,6.315,148.206
C05423=1230.919,251.653,-61.138,-176.831,6.317,148.206
C05424=1230.914,251.901,-61.165,-176.828,6.319,148.206
C05425=1230.910,252.150,-61.192,-176.826,6.321,148.205
C05426=1230.905,252.399,-61.218,-176.823,6.323,148.205
C05427=1230.901,252.647,-61.244,-176.821,6.325,148.205
C05428=1230.897,252.895,-61.272,-176.818,6.327,148.205
C05429=1230.892,253.144,-61.297,-176.816,6.329,148.204
C05430=1230.888,253.393,-61.324,-176.813,6.331,148.204
C05431=1230.883,253.641,-61.351,-176.811,6.333,148.204
C05432=1230.879,253.889,-61.378,-176.809,6.335,148.204
C05433=1230.874,254.138,-61.404,-176.806,6.337,148.203
C05434=1230.869,254.387,-61.431,-176.803,6.339,148.203
C05435=1230.866,254.635,-61.458,-176.801,6.341,148.203
C05436=1230.861,254.884,-61.485,-176.799,6.343,148.203
C05437=1230.856,255.132,-61.512,-176.796,6.345,148.202
C05438=1230.852,255.380,-61.538,-176.793,6.347,148.202
C05439=1230.847,255.629,-61.565,-176.791,6.349,148.202
C05440=1230.843,255.879,-61.592,-176.789,6.351,148.202
C05441=1230.839,256.127,-61.619,-176.786,6.353,148.201
C05442=1230.835,256.375,-61.646,-176.783,6.355,148.201
C05443=1230.830,256.624,-61.673,-176.781,6.357,148.201
C05444=1230.826,256.872,-61.699,-176.779,6.359,148.201
C05445=1230.821,257.120,-61.726,-176.776,6.361,148.200
C05446=1230.817,257.369,-61.753,-176.774,6.363,148.200
C05447=1230.812,257.618,-61.780,-176.771,6.365,148.200
C05448=1230.808,257.866,-61.806,-176.769,6.367,148.200
C05449=1230.803,258.115,-61.833,-176.766,6.369,148.199
C05450=1230.799,258.363,-61.860,-176.764,6.371,148.199
C05451=1230.794,258.612,-61.887,-176.761,6.373,148.199
C05452=1230.790,258.860,-61.914,-176.759,6.375,148.199
C05453=1230.786,259.109,-61.941,-176.757,6.377,148.199
C05454=1230.781,259.358,-61.968,-176.754,6.379,148.198
C05455=1230.777,259.606,-61.995,-176.752,6.381,148.198
C05456=1230.773,259.854,-62.022,-176.749,6.382,148.198
C05457=1230.768,260.103,-62.049,-176.747,6.385,148.198
C05458=1230.763,260.351,-62.076,-176.744,6.387,148.197
C05459=1230.759,260.600,-62.103,-176.742,6.388,148.197
C05460=1230.754,260.848,-62.130,-176.739,6.391,148.197
C05461=1230.750,261.097,-62.158,-176.737,6.393,148.197
C05462=1230.746,261.345,-62.185,-176.734,6.394,148.196
C05463=1230.742,261.594,-62.212,-176.732,6.397,148.196
C05464=1230.737,261.842,-62.239,-176.729,6.399,148.196
C05465=1230.733,262.091,-62.266,-176.726,6.401,148.196
C05466=1230.728,262.339,-62.293,-176.724,6.403,148.196
C05467=1230.723,262.588,-62.320,-176.722,6.405,148.195
C05468=1230.719,262.837,-62.347,-176.719,6.407,148.195
C05469=1230.716,263.084,-62.375,-176.717,6.409,148.195
C05470=1230.710,263.358,-62.404,-176.714,6.411,148.195
C05471=1230.705,263.630,-62.434,-176.711,6.414,148.195
C05472=1230.700,263.902,-62.464,-176.709,6.416,148.194
C05473=1230.696,264.175,-62.494,-176.706,6.418,148.194
C05474=1230.691,264.423,-62.521,-176.704,6.420,148.194
C05475=1230.687,264.672,-62.548,-176.701,6.422,148.194
C05476=1230.683,264.920,-62.576,-176.699,6.424,148.193
